SUPER^(); // FB_BA_View
Dst(); // FB_BA_BI_Raw
PlantLock(); // FB_BA_PlantLock
bPrioSfty := PlantLock.bPrioHigh OR PlantLock.bPrioLocalHigh;
bPrioCrit := PlantLock.bPrioMedium OR PlantLock.bPrioLocalMedium;
bDst := bPrioSfty OR bPrioCrit;
PrioSwiVal(
    bEn01 := stCmd.bEnSfty,
    nVal01 := stCmd.eValSfty,
    bEn02 := stCmd.bEnCrit,
    nVal02 := stCmd.eValCrit,
    bEn03 := stCmd.bEnPgm,
    nVal03 := stCmd.eValPgm); // FB_BA_PrioSwi_UDI04
MuxCmd(
    bEn := TRUE,
    nSel := PrioSwiVal.nVal,
    nEn01 := E_BA_Mdlt.eOff,
    bVal01 := FALSE,
    nEn02 := E_BA_Mdlt.eOn,
    bVal02 := TRUE,
    nEn03 := E_BA_Mdlt.eMin,
    bVal03 := TRUE,
    nEn04 := E_BA_Mdlt.eMax,
    bVal04 := TRUE); // FB_BA_MMUX_B04
Cmd(
    bEnSfty := stCmd.bEnSfty OR bPrioSfty,
    bValSfty := SEL(bPrioSfty, MuxCmd.bVal, FALSE),
    bEnCrit := stCmd.bEnCrit OR bPrioCrit,
    bValCrit := _w1,
    bEnPgm := stCmd.bEnPgm,
    bValPgm := MuxCmd.bVal); // FB_BA_BO_Raw
_w1 := SEL(bPrioCrit, MuxCmd.bVal, FALSE);
bCmd := Cmd.bPresentValue;
eActivePrio := Cmd.eActivePrio;
Ctrl(bEn := bCmd, fSetpoint := Sp.fPresentValue, fCtrlVal := fIn); // FB_BA_Loop
Sp(); // FB_BA_AV_Op
fMin := Ctrl.fMinOutputRm;
fMax := Ctrl.fMaxOutputRm;
MuxMdlt(
    bEn := bCmd,
    nSel := PrioSwiVal.nVal,
    nEn01 := E_BA_Mdlt.eOff,
    fVal01 := 0,
    nEn02 := E_BA_Mdlt.eOn,
    fVal02 := Ctrl.fPresentValue,
    nEn03 := E_BA_Mdlt.eMin,
    fVal03 := fMin,
    nEn04 := E_BA_Mdlt.eMax,
    fVal04 := fMax); // FB_BA_MMUX_R04
Mdlt(
    bEnSfty := Cmd.bEnSfty,
    fValSfty := SEL(bPrioSfty, MuxMdlt.fVal, 0),
    bEnCrit := Cmd.bEnCrit,
    fValCrit := _w2,
    bEnPgm := Cmd.bEnPgm,
    fValPgm := MuxMdlt.fVal); // FB_BA_AO_Raw
_w2 := SEL(bPrioCrit, MuxMdlt.fVal, 0);
fMdlt := Mdlt.fPresentValue;

METHOD FB_init : BOOL
VAR_INPUT
	bInitRetains : BOOL; // if TRUE, the retain variables are initialized (warm start / cold start)
	bInCopyCode : BOOL;  // if TRUE, the instance afterwards gets moved into the copy code (online change)
END_VAR
PlantLock.Parent					:= THIS^;		

Dst.iParent							:= THIS^;
Dst.iLabel							:= LblFun_Fault;  
Dst.ePolarity						:= E_BA_Polarity.eReverse;
Dst.sActiveText 					:= txtEvent_Triggered;
Dst.sInactiveText 					:= txtEvent_Normal;
Dst.nEventClassID					:= EC_ID.NC30;
Dst.stTimeDelay.nToNormal			:= BA2_Param.nDefTimeDelay_ToNormal;
Dst.stTimeDelay.nToAbnormal			:= BA2_Param.nDefTimeDelay_ToAbnormal;
Dst.bAlarmValue						:= TRUE;
Dst.aEventTransitionText[1]			:= txtEvent_Triggered;
Dst.aEventTransitionText[2]			:= txtEvent_Error;
Dst.aEventTransitionText[3]			:= txtEvent_Normal;
Dst.bEventDetectionEnable			:= TRUE;
Dst.eEnPlantLock					:= E_BA_LockPriority.eLocalMedium;

Cmd.iParent							:= THIS^;
Cmd.iLabel							:= LblFun_SwitchingCommand;  
Cmd.ePolarity						:= E_BA_Polarity.eNormal;
Cmd.sActiveText 					:= txtEvent_On;
Cmd.sInactiveText 					:= txtEvent_Off;
Cmd.bEnManualRm						:= FALSE;	//	Priority  8	
Cmd.bValManualRm					:= FALSE;	//	Priority  8
Cmd.nEventClassID					:= EC_ID.NC40;
Cmd.stTimeDelay.nToNormal			:= BA2_Param.nDefTimeDelay_ToNormal;
Cmd.stTimeDelay.nToAbnormal			:= BA2_Param.nDefTimeDelay_ToAbnormal;
Cmd.aEventTransitionText[1]			:= txtEvent_Disturb;
Cmd.aEventTransitionText[2]			:= txtEvent_None;
Cmd.aEventTransitionText[3]			:= txtEvent_Normal;
Cmd.bEventDetectionEnable			:= FALSE;
Cmd.eEnPlantLock					:= E_BA_LockPriority.eNoLock;

Mdlt.iParent						:= THIS^;
Mdlt.iLabel							:= LblFun_ControlSignal;  
Mdlt.eUnit							:= E_BA_Unit.eOther_Percent;
Mdlt.fResolution 					:= 0.003051851;
Mdlt.fScaleOffset 					:= 0;
Mdlt.fCOVIncrement					:= BA2_Param.fDefCOVIncrement;
Mdlt.bEnManualRm					:= FALSE;	//	Priority  8	
Mdlt.fValManualRm					:= 0.0;		//	Priority  8
Mdlt.nEventClassID					:= EC_ID.NC80;
Mdlt.stTimeDelay.nToNormal			:= BA2_Param.nDefTimeDelay_ToNormal;
Mdlt.stTimeDelay.nToAbnormal		:= BA2_Param.nDefTimeDelay_ToAbnormal;
Mdlt.stHighLimit.bEnable			:= FALSE;
Mdlt.stHighLimit.fValue				:= 0.0;		
Mdlt.stLowLimit.bEnable				:= FALSE;
Mdlt.stLowLimit.fValue				:= 0.0;
Mdlt.fLimitDeadband 				:= BA2_Param.fDefLimitDeadband;
Mdlt.aEventTransitionText[1]		:= txtEvent_Disturb;
Mdlt.aEventTransitionText[2]		:= txtEvent_None;
Mdlt.aEventTransitionText[3]		:= txtEvent_Normal;
Mdlt.bEventDetectionEnable			:= FALSE;
Mdlt.eEnPlantLock					:= E_BA_LockPriority.eNoLock;

Sp.iParent							:= THIS^;
Sp.iLabel							:= LblFun_Setpoint; 
Sp.eUnit 							:= E_BA_Unit.ePressure_Pascals;								 
Sp.fValueRm							:= 250;
Sp.fCOVIncrement					:= BA2_Param.fDefCOVIncrement;

Ctrl.iParent						:= THIS^;
Ctrl.iLabel							:= LblFun_LoopObject;  
Ctrl.eOpMode						:= E_BA_PIDMode.ePID;								 	 										 
Ctrl.eOutputUnit					:= E_BA_Unit.eOther_Percent;
Ctrl.eActionRm						:= E_BA_Action.eReverse;
Ctrl.fProportionalConstant			:= 0.01;
Ctrl.fIntegralConstant				:= 60;
Ctrl.fDerivativeConstant			:= 0;
Ctrl.fMaxOutputRm 					:= 100;
Ctrl.fMinOutputRm					:= 20;
Ctrl.fCOVIncrement					:= 0;
Ctrl.nDampConstant					:= 0;
Ctrl.fNeutralZone					:= 0;
END_METHOD

END_FUNCTION_BLOCK

// ---- Templates/POUs/Trade/AirConditioning/Aggregates/PreHeater/FB_BA_AC_PreHtr.TcPOU
{region '#Template'}
	{attribute 'Version' := '6.0.0.0'}
	{attribute 'Tags' := '"LCID": "1031", "Text": "AC, Aggregates, pre-heater"'}
	{attribute 'Tags' := '"LCID": "1033", "Text": "AC, Aggregates, pre-heater"'}
	{attribute 'Using' := '"Type": "Template", "URI": "Priority"'}		 
	{attribute 'Using' := '"Type": "Template", "URI": "BA2_Param"'}
	{attribute 'Using' := '"Type": "Template", "URI": "EC_ID"'}
	{attribute 'Description' := '"LCID": "1031", "Text": "Aggregat Vorerhitzer"'}
	{attribute 'Description' := '"LCID": "1033", "Text": "Aggregate pre-heater"'}
{endregion}
FUNCTION_BLOCK FB_BA_AC_PreHtr EXTENDS FB_BA_View
VAR_INPUT
	fSpTSuA					: REAL;
	fTSuA					: REAL;
	bSyncTSuACtrl			: BOOL;
	fSyncTSuACtrl			: REAL;	
	bDehumf					: BOOL;
	bSkipPreRinse			: BOOL; // Vorspülen überspringen // Skip pre-rinse
	fTWth					: REAL;
	bTWthLowLimit			: BOOL;
	bResetDehumf    		: BOOL;
END_VAR
VAR_OUTPUT
	bCmd					: BOOL;
	fPresentValue			: REAL;			
	bFrost					: BOOL;
	bPreRinseReady			: BOOL;  
	bActiveSeqCtrl			: BOOL;	
END_VAR
VAR_IN_OUT
	stTSeqLink				: ST_BA_SeqLink; // Sequenz Link Struktur // Sequence link structure	
	stAggregate				: ST_BA_Aggregate;	
END_VAR
VAR_INPUT CONSTANT PERSISTENT
	{attribute 'parameterCategory' := 'Behaviour'}
	fHysPuOn : REAL := 5.0;
	{attribute 'parameterCategory' := 'Behaviour'}
	fHysPuOff : REAL := 1.0;
END_VAR
VAR_INPUT CONSTANT
	TFl						: FB_BA_SensorAnalog;												
	TRt						: FB_BA_SensorAnalog;			
	TSuACtrl				: FB_BA_AC_PreHtrTSuACtrl;
	TRtCtrl					: FB_BA_AC_TRtCtrl;	
	TFrost					: FB_BA_SensorAnalog;																	
	TFrostPrtcCtrlAir		: FB_BA_PID_Sp;
	FrostThermostat			: FB_BA_SensorBinary;
	Vlv						: FB_BA_Vlv;
	Pu						: FB_BA_Pu1st;
	PlantLock				: FB_BA_PlantLock;			
	Aggregate				: FB_BA_Aggregate;																											 							
END_VAR
VAR
	bPrioSfty				: BOOL;
	bPrioCrit				: BOOL;		
	PrioSwiVal				: FB_BA_PrioSwi_B04;	
	
	HysPu					: FB_BA_Swi2P;
	SyncTSuACtrl			: FB_BA_RFTrig;
	SyncSeqCtrlIsActive		: FB_BA_RFTrig;
	PrioSwiSync				: FB_BA_PrioSwi_R04;	
END_VAR
VAR // added by the converter: edge detectors and wires of the graphical bodies
    _s1 : ST_BA_Analog;
    _s2 : ST_BA_Binary;
    _w1 : ANY;
    _w2 : BOOL;
END_VAR

SUPER^(); // FB_BA_View
Aggregate(bFdbUp := bPreRinseReady, stAggregate := stAggregate); // FB_BA_Aggregate
PlantLock(); // FB_BA_PlantLock
bPrioSfty := PlantLock.bPrioHigh OR PlantLock.bPrioLocalHigh;
bPrioCrit := PlantLock.bPrioMedium OR PlantLock.bPrioLocalMedium;
TFl(); // FB_BA_SensorAnalog
TRt(); // FB_BA_SensorAnalog
PrioSwiVal(
    bEn01 := Aggregate.arrPriorities[Priority.nLifeSafety],
    bVal01 := Aggregate.bValue,
    bEn02 := Aggregate.arrPriorities[Priority.nCritical],
    bVal02 := Aggregate.bValue,
    bEn03 := Aggregate.arrPriorities[Priority.nProgram],
    bVal03 := Aggregate.bValue); // FB_BA_PrioSwi_B04
SyncTSuACtrl(bValue := bSyncTSuACtrl); // FB_BA_RFTrig
SyncSeqCtrlIsActive(bValue := TSuACtrl.bSeqActv); // FB_BA_RFTrig
PrioSwiSync(
    bEn01 := SyncTSuACtrl.Qr,
    fVal01 := fSyncTSuACtrl,
    bEn04 := SyncSeqCtrlIsActive.Qr AND bActiveSeqCtrl AND bTWthLowLimit,
    fVal04 := Vlv.fMdlt); // FB_BA_PrioSwi_R04
TSuACtrl(
    bEn := PrioSwiVal.bVal,
    fSpTSuA := fSpTSuA,
    fTSuA := fTSuA,
    bSync := PrioSwiSync.bQ,
    fSync := PrioSwiSync.fVal,
    bDehumf := bDehumf,
    bResetDehumf := bResetDehumf,
    stSeqLink := stTSeqLink); // FB_BA_AC_PreHtrTSuACtrl
bActiveSeqCtrl := TSuACtrl.bIsActive;
TRtCtrl(
    bEnPreRinse := PrioSwiVal.bVal,
    fTRt := TRt.fPresentValue,
    bTWthLowLimit := bTWthLowLimit,
    fTWth := fTWth,
    bSkipPreRinse := bSkipPreRinse,
    bSeqActive := stTSeqLink.bEnSeqLink); // FB_BA_AC_TRtCtrl
bPreRinseReady := TRtCtrl.bPreRinseReady;
TFrost(); // FB_BA_SensorAnalog
TFrostPrtcCtrlAir(bEn := TRUE, fX := TFrost.fPresentValue); // FB_BA_PID_Sp
FrostThermostat(); // FB_BA_SensorBinary
bFrost := TFrost.eEventState = E_BA_EventState.eLowLimit OR FrostThermostat.bPresentValue;
_w1 := MAX(TSuACtrl.fY, TRtCtrl.fY, TFrostPrtcCtrlAir.fY);
// compose _s1 : ST_BA_Analog
_s1.bEnSfty := Aggregate.arrPriorities[Priority.nLifeSafety] OR bPrioSfty;
_s1.fValSfty := _w1;
_s1.bEnCrit := Aggregate.arrPriorities[Priority.nCritical] OR bPrioCrit OR bFrost;
_s1.fValCrit := SEL(bFrost, _w1, 100);
_s1.bEnPgm := TRUE;
_s1.fValPgm := _w1;
Vlv(stCmd := _s1); // FB_BA_Vlv
fPresentValue := Vlv.fMdlt;
HysPu(bEn := TRUE, fIn := fPresentValue, fOn := fHysPuOn, fOff := fHysPuOff); // FB_BA_Swi2P
_w2 := HysPu.bQ OR bTWthLowLimit OR bFrost;
// compose _s2 : ST_BA_Binary
_s2.bEnSfty := Vlv.stCmd.bEnSfty;
_s2.bValSfty := _w2;
_s2.bEnCrit := Vlv.stCmd.bEnCrit;
_s2.bValCrit := _w2;
_s2.bEnPgm := TRUE;
_s2.bValPgm := _w2;
Pu(stCmd := _s2); // FB_BA_Pu1st
bCmd := Pu.bCmd;

METHOD FB_init : BOOL
VAR_INPUT
	bInitRetains : BOOL; // if TRUE, the retain variables are initialized (warm start / cold start)
	bInCopyCode : BOOL;  // if TRUE, the instance afterwards gets moved into the copy code (online change)
END_VAR
PlantLock.Parent								:= THIS^;		

TFl.iParent										:= THIS^;		
TFl.iLabel										:= LblAgg_TemperatureFlow;   
TFl.sObjectName									:= '{Idx=11}';						 
TFl.eDPADMode									:= E_BA_DPADMode.eInclude;
TFl.MV.eUnit									:= E_BA_Unit.eTemperature_DegreesCelsius;
TFl.MV.fResolution 								:= 0.01;
TFl.MV.fScaleOffset 							:= 0; 
TFl.MV.bEventDetectionEnable					:= TRUE;
TFl.MV.eEnPlantLock								:= E_BA_LockPriority.eNoLock;
                            					                            					
TRt.iParent										:= THIS^;		
TRt.iLabel										:= LblAgg_TemperatureReturnFlow;   
TRt.sObjectName									:= '{Idx=11}';						 
TRt.eDPADMode									:= E_BA_DPADMode.eInclude;
TRt.MV.eUnit									:= E_BA_Unit.eTemperature_DegreesCelsius;
TRt.MV.fResolution 								:= 0.01;
TRt.MV.fScaleOffset 							:= 0;  
TRt.MV.bEventDetectionEnable					:= TRUE;
TRt.MV.eEnPlantLock								:= E_BA_LockPriority.eMedium;

TSuACtrl.iParent								:= THIS^;	
TSuACtrl.iLabel									:= LblCtl_SupplyAirTemperatureControl;   
TSuACtrl.sObjectName							:= '{Idx=11}';						 
TSuACtrl.eDPADMode								:= E_BA_DPADMode.eInclude;								

TRtCtrl.iParent									:= THIS^;
TRtCtrl.iLabel									:= LblCtl_ReturnWaterControl;   
TRtCtrl.sObjectName								:= '{Idx=12}';						 
TRtCtrl.eDPADMode								:= E_BA_DPADMode.eInclude;								
TRtCtrl.PreRinseDst.bEventDetectionEnable		:= TRUE;
TRtCtrl.PreRinseDst.eEnPlantLock				:= E_BA_LockPriority.eNoLock;
	                                				
TFrost.iParent									:= THIS^;		
TFrost.iLabel									:= LblCtl_TemperatureFrost;   
TFrost.sObjectName								:= '{Idx=11}';						 
TFrost.eDPADMode								:= E_BA_DPADMode.eInclude;
TFrost.MV.eUnit									:= E_BA_Unit.eTemperature_DegreesCelsius;
TFrost.MV.fResolution 							:= 0.0004577776;
TFrost.MV.fScaleOffset 							:= 0;  
TFrost.MV.bEventDetectionEnable					:= TRUE;
TFrost.MV.eEnPlantLock							:= E_BA_LockPriority.eMedium;

TFrostPrtcCtrlAir.iParent						:= THIS^;	
TFrostPrtcCtrlAir.iLabel						:= LblCtl_FrostProtectionControl;   
TFrostPrtcCtrlAir.sObjectName					:= '{Idx=13}';						 
TFrostPrtcCtrlAir.eDPADMode						:= E_BA_DPADMode.eInclude;
TFrostPrtcCtrlAir.Sp.fValueRm 					:= 5.0;
TFrostPrtcCtrlAir.Ctrl.fProportionalConstant	:= 5;
TFrostPrtcCtrlAir.Ctrl.fIntegralConstant		:= 60;	
TFrostPrtcCtrlAir.Ctrl.eActionRm				:= E_BA_Action.eReverse;

FrostThermostat.iParent							:= THIS^; 
FrostThermostat.iLabel							:= LblAgg_FrostProtectionMonitor;   
FrostThermostat.sObjectName						:= '{Idx=13}';						 
FrostThermostat.eDPADMode						:= E_BA_DPADMode.eInclude;
FrostThermostat.Input.iLabel					:= LblFun_OperationalMessage;   
FrostThermostat.Input.sObjectName				:= '{Idx=13}';						 
FrostThermostat.Input.ePolarity					:= E_BA_Polarity.eReverse;
FrostThermostat.Input.sActiveText 				:= txtEvent_Triggered;
FrostThermostat.Input.sInactiveText 			:= txtEvent_Normal;
FrostThermostat.Input.nEventClassID				:= EC_ID.NC30;
FrostThermostat.Input.aEventTransitionText[1]	:= txtEvent_Triggered;
FrostThermostat.Input.aEventTransitionText[2]	:= txtEvent_Error;
FrostThermostat.Input.aEventTransitionText[3]	:= txtEvent_Normal;
FrostThermostat.Input.bEventDetectionEnable		:= TRUE;
FrostThermostat.Input.eEnPlantLock				:= E_BA_LockPriority.eMedium;	

Vlv.iParent										:= THIS^;
Vlv.iLabel										:= LblAgg_Valve;    									 
Vlv.sObjectName									:= '{Idx=11}';						 
Vlv.eDPADMode									:= E_BA_DPADMode.eInclude;								
                            					
Pu.iParent										:= THIS^;
Pu.iLabel										:= LblAgg_Pump;   									 
Pu.sObjectName									:= '{Idx=11}';						 
Pu.eDPADMode									:= E_BA_DPADMode.eInclude;
Pu.Dst.bEventDetectionEnable					:= TRUE;
Pu.Dst.eEnPlantLock								:= E_BA_LockPriority.eMedium;
END_METHOD

END_FUNCTION_BLOCK

// ---- Templates/POUs/Universal/Pump/1st/FB_BA_Pu1st.TcPOU
{region '#Template'}
	{attribute 'Version' := '5.0.0.0'}
	{attribute 'Tags' := '"LCID": "1031", "Text": "Universal, Pump"'}
	{attribute 'Tags' := '"LCID": "1033", "Text": "Universal, Pump"'}
	{attribute 'Using' := '"Type": "Template", "URI": "EC_ID"'}
	{attribute 'Using' := '"Type": "Template", "URI": "BA2_Param"'}
	{attribute 'Description' := '"LCID": "1031", "Text": "Pumpe 1 stufig"'}
	{attribute 'Description' := '"LCID": "1033", "Text": "Pump 1 stage"'}
{endregion}	 
FUNCTION_BLOCK FB_BA_Pu1st EXTENDS FB_BA_Mot1st
VAR_INPUT
	bAblkLock				: BOOL;	
END_VAR
VAR_INPUT CONSTANT
	DlyOff					: FB_BA_DlyOff;								
	Ablk					: FB_BA_AntiBlocking;							
END_VAR
VAR
	PrioSwiPgm				: FB_BA_PrioSwi_B04;
	tonAblkLock				: TON;
END_VAR
VAR // added by the converter: edge detectors and wires of the graphical bodies
    _s1 : ST_BA_Binary;
END_VAR

DlyOff(bVal := stCmd.bEnPgm AND stCmd.bValPgm); // FB_BA_DlyOff
tonAblkLock(IN := bAblkLock, PT := T#2s); // TON
Ablk(bFdb := bCmd, bLock := tonAblkLock.Q); // FB_BA_AntiBlocking
PrioSwiPgm(bEn03 := DlyOff.bQ, bVal03 := TRUE, bEn04 := Ablk.bQ, bVal04 := TRUE); // FB_BA_PrioSwi_B04
// compose _s1 : ST_BA_Binary
_s1.bEnSfty := stCmd.bEnSfty;
_s1.bValSfty := stCmd.bValSfty;
_s1.bEnCrit := stCmd.bEnCrit;
_s1.bValCrit := stCmd.bValCrit;
_s1.bEnPgm := PrioSwiPgm.bQ;
_s1.bValPgm := PrioSwiPgm.bVal;
SUPER^(stCmd := _s1); // FB_BA_Mot1st

METHOD FB_init : BOOL
VAR_INPUT
	bInitRetains : BOOL; // if TRUE, the retain variables are initialized (warm start / cold start)
	bInCopyCode : BOOL;  // if TRUE, the instance afterwards gets moved into the copy code (online change)
END_VAR
DlyOff.iParent			:= THIS^;	
DlyOff.iLabel			:= LblCtl_DelayOff;
DlyOff.eDPADMode		:= E_BA_DPADMode.eIncludeDescription;

Ablk.iParent			:= THIS^;	 
Ablk.iLabel				:= LblCtl_AntiBlocking;
Ablk.eDPADMode			:= E_BA_DPADMode.eIncludeDescription;
END_METHOD

END_FUNCTION_BLOCK

// ---- Templates/POUs/Trade/AirConditioning/General/FB_BA_AC_OpMod1St.TcPOU
{region '#Template'}
	{attribute 'Version' := '6.0.0.0'}
	{attribute 'Tags' := '"LCID": "1031", "Text": "AC, Allgemein, AHU, Betriebsart"'}
	{attribute 'Tags' := '"LCID": "1033", "Text": "AC, General, AHU, Operating mode"'}
	{attribute 'Using' := '"Type": "Template", "URI": "E_BA_AC_OpMod01"'}
	{attribute 'Using' := '"Type": "Template", "URI": "E_BA_OnOffA"'}
	{attribute 'Using' := '"Type": "Template", "URI": "E_BA_OnOff"'}
	{attribute 'Description' := '"LCID": "1031", "Text": "Betriebsart"'}
	{attribute 'Description' := '"LCID": "1033", "Text": "Operating mode"'}
{endregion}
FUNCTION_BLOCK FB_BA_AC_OpMod1St EXTENDS FB_BA_View
VAR_INPUT
	bSmExtt					: BOOL;	// smoke extraction 
	bFireDetc				: BOOL;	// fire detection alarm
	bForcVent				: BOOL;	// Forced ventilation
	bEmgOff					: BOOL;	// emergency stop
	bFrst					: BOOL;	// Frost protection is active
	bCentSwiOff				: BOOL;	// Central switch-off	
	bAlmShutOff				: BOOL;	// Shut Off plant collective alarm
	bNgtCol					: BOOL;	// Summer night cooling
	bColDwnPrtc				: BOOL;	// Cooling down protection
	bOvrHtgPrtc				: BOOL;	// Overheating protection
END_VAR
VAR_OUTPUT
	eOpMode					: E_BA_AC_OpMod01;
END_VAR
VAR_INPUT CONSTANT
	OpModMan				: FB_BA_MV_Op;	
	Sched					: FB_BA_SchedM;
	OpModPr					: FB_BA_MV_Op;
END_VAR
VAR
	PrioSwiOpMod			: FB_BA_PrioSwi_UDI24;
END_VAR

SUPER^(); // FB_BA_View
OpModMan(); // FB_BA_MV_Op
Sched(); // FB_BA_SchedM
PrioSwiOpMod(
    bEn02 := bSmExtt,
    nVal02 := E_BA_AC_OpMod01.eSmokeExtractionProgram,
    bEn04 := bFireDetc,
    nVal04 := E_BA_AC_OpMod01.eFire,
    bEn05 := bCentSwiOff,
    nVal05 := E_BA_AC_OpMod01.eCentralSwitchOff,
    bEn07 := bForcVent,
    nVal07 := E_BA_AC_OpMod01.eForcedVentilation,
    bEn08 := bEmgOff,
    nVal08 := E_BA_AC_OpMod01.eEmergency,
    bEn09 := bFrst,
    nVal09 := E_BA_AC_OpMod01.eFrost,
    bEn10 := bAlmShutOff,
    nVal10 := E_BA_AC_OpMod01.eAlarm,
    bEn14 := E_BA_OnOffA.eOff = OpModMan.nPresentValue,
    nVal14 := E_BA_AC_OpMod01.eOff,
    bEn15 := OpModMan.nPresentValue = E_BA_OnOffA.eOn,
    nVal15 := E_BA_AC_OpMod01.eOn,
    bEn18 := Sched.nPresentValue = E_BA_OnOff.eOn,
    nVal18 := E_BA_AC_OpMod01.eOn,
    bEn20 := bNgtCol,
    nVal20 := E_BA_AC_OpMod01.eNightCooling,
    bEn21 := bColDwnPrtc,
    nVal21 := E_BA_AC_OpMod01.eCoolDownProtection,
    bEn22 := bOvrHtgPrtc,
    nVal22 := E_BA_AC_OpMod01.eOverHeatingProtection,
    bEn24 := TRUE,
    nVal24 := E_BA_AC_OpMod01.eOFF); // FB_BA_PrioSwi_UDI24
OpModPr(nValuePgm := PrioSwiOpMod.nVal); // FB_BA_MV_Op
eOpMode := OpModPr.nPresentValue;

METHOD FB_init : BOOL
VAR_INPUT
	bInitRetains : BOOL; // if TRUE, the retain variables are initialized (warm start / cold start)
	bInCopyCode : BOOL;  // if TRUE, the instance afterwards gets moved into the copy code (online change)
END_VAR
OpModMan.iParent			:= THIS^;
OpModMan.iLabel				:= LblCtl_OperationModeSelection; 	
OpModMan.aStateText[1]		:= txtEvent_Auto;
OpModMan.aStateText[2]		:= txtEvent_Off;
OpModMan.aStateText[3]		:= txtEvent_On;
OpModMan.nValueRm			:= E_BA_OnOffA.eAutomatic;

OpModPr.iParent				:= THIS^;
OpModPr.iLabel				:= LblCtl_PresentOperationMode; 								 	 
OpModPr.aStateText[1]		:= txtEvent_Off;
OpModPr.aStateText[2]		:= txtEvent_On;
OpModPr.aStateText[3]		:= txtEvent_EmergencyStop;
OpModPr.aStateText[4]		:= txtEvent_Frost;
OpModPr.aStateText[5]		:= txtEvent_SmokeExtraction_P;
OpModPr.aStateText[6]		:= txtEvent_SmokeExtractionSupplyAir;
OpModPr.aStateText[7]		:= txtEvent_SmokeExtractionExtractAir;
OpModPr.aStateText[8]		:= txtEvent_Fire;
OpModPr.aStateText[9]		:= txtEvent_NightCooling;
OpModPr.aStateText[10]		:= txtEvent_CoolDownProtection;
OpModPr.aStateText[11]		:= txtEvent_OverHeatingProtection;
OpModPr.aStateText[12]		:= txtEvent_Disturb;
OpModPr.aStateText[13]		:= txtEvent_ForcedVentilation;
OpModPr.aStateText[14]		:= txtEvent_CentralSwitchOff; 		

Sched.iParent											:= THIS^;
Sched.iLabel											:= LblFun_Scheduler; 			
Sched.aStateText[1]										:= txtEvent_Off;
Sched.aStateText[2]										:= txtEvent_On;
Sched.nPredictTime										:= 0;
Sched.nDefaultValue										:= E_BA_OnOff.eOff;
Sched.bWriteWeekly										:= FALSE;
//	Monday
Sched.aWeek[E_BA_Weekday.eMonday,1].eState				:= E_BA_SchedEntryState.eValue;
Sched.aWeek[E_BA_Weekday.eMonday,1].uValue.udiVal		:= E_BA_OnOff.eOn;
Sched.aWeek[E_BA_Weekday.eMonday,1].stTime.nHour		:= 6;
Sched.aWeek[E_BA_Weekday.eMonday,1].stTime.nMinute		:= 0;
Sched.aWeek[E_BA_Weekday.eMonday,1].stTime.nSecond		:= 0;
Sched.aWeek[E_BA_Weekday.eMonday,2].eState				:= E_BA_SchedEntryState.eValue;
Sched.aWeek[E_BA_Weekday.eMonday,2].uValue.udiVal		:= E_BA_OnOff.eOff;
Sched.aWeek[E_BA_Weekday.eMonday,2].stTime.nHour		:= 20;
Sched.aWeek[E_BA_Weekday.eMonday,2].stTime.nMinute		:= 0;
Sched.aWeek[E_BA_Weekday.eMonday,2].stTime.nSecond		:= 0;
Sched.aWeek[E_BA_Weekday.eMonday,3].eState				:= E_BA_SchedEntryState.eValue;
Sched.aWeek[E_BA_Weekday.eMonday,3].uValue.udiVal		:= E_BA_OnOff.eOff;
Sched.aWeek[E_BA_Weekday.eMonday,3].stTime.nHour		:= 0;
Sched.aWeek[E_BA_Weekday.eMonday,3].stTime.nMinute		:= 0;
Sched.aWeek[E_BA_Weekday.eMonday,3].stTime.nSecond		:= 0;
//	Tuesday
Sched.aWeek[E_BA_Weekday.eTuesday,1].eState				:= E_BA_SchedEntryState.eValue;
Sched.aWeek[E_BA_Weekday.eTuesday,1].uValue.udiVal		:= E_BA_OnOff.eOn;
Sched.aWeek[E_BA_Weekday.eTuesday,1].stTime.nHour		:= 6;
Sched.aWeek[E_BA_Weekday.eTuesday,1].stTime.nMinute		:= 0;
Sched.aWeek[E_BA_Weekday.eTuesday,1].stTime.nSecond		:= 0;
Sched.aWeek[E_BA_Weekday.eTuesday,2].eState				:= E_BA_SchedEntryState.eValue;
Sched.aWeek[E_BA_Weekday.eTuesday,2].uValue.udiVal		:= E_BA_OnOff.eOff;
Sched.aWeek[E_BA_Weekday.eTuesday,2].stTime.nHour		:= 20;
Sched.aWeek[E_BA_Weekday.eTuesday,2].stTime.nMinute		:= 0;
Sched.aWeek[E_BA_Weekday.eTuesday,2].stTime.nSecond		:= 0;
Sched.aWeek[E_BA_Weekday.eTuesday,3].eState				:= E_BA_SchedEntryState.eValue;
Sched.aWeek[E_BA_Weekday.eTuesday,3].uValue.udiVal		:= E_BA_OnOff.eOff;
Sched.aWeek[E_BA_Weekday.eTuesday,3].stTime.nHour		:= 0;
Sched.aWeek[E_BA_Weekday.eTuesday,3].stTime.nMinute		:= 0;
Sched.aWeek[E_BA_Weekday.eTuesday,3].stTime.nSecond		:= 0;
//	Wednesday
Sched.aWeek[E_BA_Weekday.eWednesday,1].eState			:= E_BA_SchedEntryState.eValue;
Sched.aWeek[E_BA_Weekday.eWednesday,1].uValue.udiVal	:= E_BA_OnOff.eOn;
Sched.aWeek[E_BA_Weekday.eWednesday,1].stTime.nHour		:= 6;
Sched.aWeek[E_BA_Weekday.eWednesday,1].stTime.nMinute	:= 0;
Sched.aWeek[E_BA_Weekday.eWednesday,1].stTime.nSecond	:= 0;
Sched.aWeek[E_BA_Weekday.eWednesday,2].eState			:= E_BA_SchedEntryState.eValue;
Sched.aWeek[E_BA_Weekday.eWednesday,2].uValue.udiVal	:= E_BA_OnOff.eOff;
Sched.aWeek[E_BA_Weekday.eWednesday,2].stTime.nHour		:= 20;
Sched.aWeek[E_BA_Weekday.eWednesday,2].stTime.nMinute	:= 0;
Sched.aWeek[E_BA_Weekday.eWednesday,2].stTime.nSecond	:= 0;
Sched.aWeek[E_BA_Weekday.eWednesday,3].eState			:= E_BA_SchedEntryState.eValue;
Sched.aWeek[E_BA_Weekday.eWednesday,3].uValue.udiVal	:= E_BA_OnOff.eOff;
Sched.aWeek[E_BA_Weekday.eWednesday,3].stTime.nHour		:= 0;
Sched.aWeek[E_BA_Weekday.eWednesday,3].stTime.nMinute	:= 0;
Sched.aWeek[E_BA_Weekday.eWednesday,3].stTime.nSecond	:= 0;
//	Thursday
Sched.aWeek[E_BA_Weekday.eThursday,1].eState			:= E_BA_SchedEntryState.eValue;
Sched.aWeek[E_BA_Weekday.eThursday,1].uValue.udiVal		:= E_BA_OnOff.eOn;
Sched.aWeek[E_BA_Weekday.eThursday,1].stTime.nHour		:= 6;
Sched.aWeek[E_BA_Weekday.eThursday,1].stTime.nMinute	:= 0;
Sched.aWeek[E_BA_Weekday.eThursday,1].stTime.nSecond	:= 0;
Sched.aWeek[E_BA_Weekday.eThursday,2].eState			:= E_BA_SchedEntryState.eValue;
Sched.aWeek[E_BA_Weekday.eThursday,2].uValue.udiVal		:= E_BA_OnOff.eOff;
Sched.aWeek[E_BA_Weekday.eThursday,2].stTime.nHour		:= 20;
Sched.aWeek[E_BA_Weekday.eThursday,2].stTime.nMinute	:= 0;
Sched.aWeek[E_BA_Weekday.eThursday,2].stTime.nSecond	:= 0;
Sched.aWeek[E_BA_Weekday.eThursday,3].eState			:= E_BA_SchedEntryState.eValue;
Sched.aWeek[E_BA_Weekday.eThursday,3].uValue.udiVal		:= E_BA_OnOff.eOff;
Sched.aWeek[E_BA_Weekday.eThursday,3].stTime.nHour		:= 0;
Sched.aWeek[E_BA_Weekday.eThursday,3].stTime.nMinute	:= 0;
Sched.aWeek[E_BA_Weekday.eThursday,3].stTime.nSecond	:= 0;
//	Friday
Sched.aWeek[E_BA_Weekday.eFriday,1].eState				:= E_BA_SchedEntryState.eValue;
Sched.aWeek[E_BA_Weekday.eFriday,1].uValue.udiVal		:= E_BA_OnOff.eOn;
Sched.aWeek[E_BA_Weekday.eFriday,1].stTime.nHour		:= 6;
Sched.aWeek[E_BA_Weekday.eFriday,1].stTime.nMinute		:= 0;
Sched.aWeek[E_BA_Weekday.eFriday,1].stTime.nSecond		:= 0;
Sched.aWeek[E_BA_Weekday.eFriday,2].eState				:= E_BA_SchedEntryState.eValue;
Sched.aWeek[E_BA_Weekday.eFriday,2].uValue.udiVal		:= E_BA_OnOff.eOff;
Sched.aWeek[E_BA_Weekday.eFriday,2].stTime.nHour		:= 20;
Sched.aWeek[E_BA_Weekday.eFriday,2].stTime.nMinute		:= 0;
Sched.aWeek[E_BA_Weekday.eFriday,2].stTime.nSecond		:= 0;
Sched.aWeek[E_BA_Weekday.eFriday,3].eState				:= E_BA_SchedEntryState.eValue;
Sched.aWeek[E_BA_Weekday.eFriday,3].uValue.udiVal		:= E_BA_OnOff.eOff;
Sched.aWeek[E_BA_Weekday.eFriday,3].stTime.nHour		:= 0;
Sched.aWeek[E_BA_Weekday.eFriday,3].stTime.nMinute		:= 0;
Sched.aWeek[E_BA_Weekday.eFriday,3].stTime.nSecond		:= 0;
Sched.bWriteException									:= FALSE;
END_METHOD

END_FUNCTION_BLOCK

// ---- Templates/POUs/Trade/AutomationControl/ControlCabinet/FB_BA_ControlCabinet.TcPOU
{region '#Template'}
	{attribute 'Version' := '5.0.1.0'}
	{attribute 'Tags' := '"LCID": "1031", "Text": "General, Cabinet, Control cabinet"'}
	{attribute 'Tags' := '"LCID": "1033", "Text": "General, Cabinet, Control cabinet"'}
	{attribute 'Using' := '"Type": "Template", "URI": "EC_ID"'}
	{attribute 'Description' := '"LCID": "1031", "Text": "Schaltschrank Ereignisse"'}
	{attribute 'Description' := '"LCID": "1033", "Text": "Control cabinet events"'}
{endregion}
FUNCTION_BLOCK FB_BA_ControlCabinet EXTENDS FB_BA_ControlCabinetBasic
VAR_INPUT CONSTANT
	Fuse01					: FB_BA_SensorBinary;		
	Fuse02					: FB_BA_SensorBinary;	
	Fuse03					: FB_BA_SensorBinary;	
END_VAR

SUPER^(); // FB_BA_ControlCabinetBasic
Fuse01(); // FB_BA_SensorBinary
Fuse02(); // FB_BA_SensorBinary
Fuse03(); // FB_BA_SensorBinary

METHOD FB_init : BOOL
VAR_INPUT
	bInitRetains : BOOL; // if TRUE, the retain variables are initialized (warm start / cold start)
	bInCopyCode : BOOL;  // if TRUE, the instance afterwards gets moved into the copy code (online change)
END_VAR
Fuse01.iParent								:= THIS^;
Fuse01.iLabel								:= LblCtl_Fuse;
Fuse01.sObjectName							:='{Idx=10}';	
Fuse01.eDPADMode							:= E_BA_DPADMode.eInclude;	
Fuse01.Input.iLabel							:= LblFun_Fault;																																									
Fuse01.Input.ePolarity						:= E_BA_Polarity.eReverse;
Fuse01.Input.sActiveText 					:= txtEvent_Triggered;
Fuse01.Input.sInactiveText 					:= txtEvent_Normal;
Fuse01.Input.nEventClassID					:= EC_ID.NC30;
Fuse01.Input.aEventTransitionText[1]		:= txtEvent_Triggered;
Fuse01.Input.aEventTransitionText[2]		:= txtEvent_Error;
Fuse01.Input.aEventTransitionText[3]		:= txtEvent_Normal;
Fuse01.Input.bEventDetectionEnable			:= TRUE;

Fuse01.Input.eEnPlantLock					:= E_BA_LockPriority.eNoLock;	
								 
Fuse02.iParent								:= THIS^;		
Fuse02.iLabel								:= LblCtl_Fuse;	
Fuse02.sObjectName							:='{Idx=20}';	
Fuse02.eDPADMode							:= E_BA_DPADMode.eInclude;	
Fuse02.Input.iLabel							:= LblFun_Fault;																				
Fuse02.Input.ePolarity						:= E_BA_Polarity.eReverse;
Fuse02.Input.sActiveText 					:= txtEvent_Triggered;
Fuse02.Input.sInactiveText 					:= txtEvent_Normal;
Fuse02.Input.nEventClassID					:= EC_ID.NC30;
Fuse02.Input.aEventTransitionText[1]		:= txtEvent_Triggered;
Fuse02.Input.aEventTransitionText[2]		:= txtEvent_Error;
Fuse02.Input.aEventTransitionText[3]		:= txtEvent_Normal;
Fuse02.Input.bEventDetectionEnable			:= TRUE;

Fuse02.Input.eEnPlantLock					:= E_BA_LockPriority.eNoLock;	
										 
Fuse03.iParent								:= THIS^;		
Fuse03.iLabel								:= LblCtl_Fuse;	
Fuse03.sObjectName							:='{Idx=30}';	
Fuse03.eDPADMode							:= E_BA_DPADMode.eInclude;				
Fuse03.Input.iLabel							:= LblFun_Fault;																				
Fuse03.Input.ePolarity						:= E_BA_Polarity.eReverse;
Fuse03.Input.sActiveText 					:= txtEvent_Triggered;
Fuse03.Input.sInactiveText 					:= txtEvent_Normal;
Fuse03.Input.nEventClassID					:= EC_ID.NC30;
Fuse03.Input.aEventTransitionText[1]		:= txtEvent_Triggered;
Fuse03.Input.aEventTransitionText[2]		:= txtEvent_Error;
Fuse03.Input.aEventTransitionText[3]		:= txtEvent_Normal;
Fuse03.Input.bEventDetectionEnable			:= TRUE;

Fuse03.Input.eEnPlantLock					:= E_BA_LockPriority.eNoLock;
END_METHOD

END_FUNCTION_BLOCK

// ---- Templates/POUs/Trade/AutomationControl/Device/FB_BA_Device.TcPOU
{region '#Template'}
	{attribute 'Version' := '5.0.1.0'}
	{attribute 'Tags' := '"LCID": "1031", "Text": "Automatisierungssteuerung, Gerät, Einstellungen, Projekt, Parameter, Trend, Empfängerliste"'}
	{attribute 'Tags' := '"LCID": "1033", "Text": "Automation control, Device, Settings, Project, Parameter, Trend, Recipient list"'}
	{attribute 'Description' := '"LCID": "1031", "Text": "Basis Einstellungen der Steuerung"'}
	{attribute 'Description' := '"LCID": "1033", "Text": "Basic settings of the control"'}
{endregion}
	 
FUNCTION_BLOCK FB_BA_Device EXTENDS FB_BA_View
VAR_INPUT
END_VAR
VAR_INPUT CONSTANT
	Trend				: FB_BA_TrendLogging;	
	Project				: FB_BA_ProjectEx;
	Parameter			: FB_BA_Parameter;	
END_VAR
VAR_OUTPUT
END_VAR
VAR
	tonDlyStartPLC		: TON;	
END_VAR

SUPER^(); // FB_BA_View
tonDlyStartPLC(IN := TRUE, PT := T#2000ms); // TON
BA2_Param.bDlyStartPLC := tonDlyStartPLC.Q;
Parameter(); // FB_BA_Parameter
Trend(); // FB_BA_TrendLogging
// connect a UPS-monitoring FB at this input
Project(); // FB_BA_ProjectEx

METHOD FB_init : BOOL
VAR_INPUT
	bInitRetains : BOOL; // if TRUE, the retain variables are initialized (warm start / cold start)
	bInCopyCode : BOOL;  // if TRUE, the instance afterwards gets moved into the copy code (online change)
END_VAR
Project.iParent						:= THIS^;
Project.iLabel						:= LblComp_Project;
Project.sObjectName					:= '{Idx=11,Idx=99}';
Project.tPrsData_DefaultPeriod 		:= T#30M;
Project.tPrsData_ComissioningPeriod := T#10M;

Trend.iParent						:= THIS^;
Trend.iLabel						:= LblCtl_TrendLogging;
Trend.eDPADMode						:= E_BA_DPADMode.eInclude;
END_METHOD

END_FUNCTION_BLOCK

// ---- Templates/POUs/Universal/Control/Trend/FB_BA_TrendLogging.TcPOU
{region '#Template'}
	{attribute 'Version' := '5.0.1.0'}
	{attribute 'Tags' := '"LCID": "1031", "Text": "Universal, Control, Trend"'}
	{attribute 'Tags' := '"LCID": "1033", "Text": "Universal, Control, Trend"'}
	{attribute 'Using' := '"Type": "Template", "URI": "EC_ID"'}
	{attribute 'Using' := '"Type": "Template", "URI": "BA2_Param"'}
	{attribute 'Description' := '"LCID": "1031", "Text": "Trend"'}
	{attribute 'Description' := '"LCID": "1033", "Text": "Trend"'}
{endregion}			 
FUNCTION_BLOCK FB_BA_TrendLogging EXTENDS FB_BA_View
VAR_INPUT
END_VAR
VAR_OUTPUT
END_VAR
VAR_INPUT CONSTANT
	Trends						: ARRAY[1..TREND_COUNT] OF FB_BA_Trend;								
END_VAR
VAR
	i							: UDINT;
END_VAR
VAR CONSTANT
	TREND_COUNT						: UDINT := 30;
END_VAR

SUPER^();

FOR i := 1 TO TREND_COUNT DO
	Trends[i]();
END_FOR

METHOD FB_init : BOOL
VAR_INPUT
	bInitRetains : BOOL; // if TRUE, the retain variables are initialized (warm start / cold start)
	bInCopyCode : BOOL;  // if TRUE, the instance afterwards gets moved into the copy code (online change)
END_VAR 
VAR
END_VAR
FOR i := 1 TO TREND_COUNT DO
	Trends[i].iParent					:= THIS^;
	Trends[i].iLabel					:= LblFun_ObjectTrendLog;
	Trends[i].bEnable					:= BA2_Param.bTrend_DefLogEnable;
	Trends[i].stStartTime				:= BA2_Param.stTrend_DefStartTime;
	Trends[i].stStopTime				:= BA2_Param.stTrend_DefStopTime;	
	Trends[i].nLogInterval 				:= BA2_Param.nTrend_DefLogInterval;
	Trends[i].bStopOnFull				:= BA2_Param.bTrend_DefStopOnFull;
	Trends[i].nBufferSize 				:= BA2_Param.nTrend_BufferSize;
	Trends[i].eLoggingType				:= BA2_Param.eTrend_DefLoggingType;	
	Trends[i].nEventClassID				:= EC_ID.NC80;
	Trends[i].nNotificationThreshold	:= BA2_Param.nTrend_DefNotificationThreshold;
	Trends[i].aEventTransitionText[1]	:= txtEvent_Offnormal;
	Trends[i].aEventTransitionText[2]	:= txtEvent_None;
	Trends[i].aEventTransitionText[3]	:= txtEvent_Normal;
	Trends[i].bEventDetectionEnable		:= FALSE;
END_FOR
END_METHOD

END_FUNCTION_BLOCK

// ---- Templates/POUs/Trade/AutomationControl/Device/Project/FB_BA_ProjectEx.TcPOU
{region '#Template'}
	{attribute 'Version' := '5.0.0.0'}
	{attribute 'Tags' := '"LCID": "1031", "Text": "Automatisierungssteuerung, Gerät, Einstellungen, Projekt"'}
	{attribute 'Tags' := '"LCID": "1033", "Text": "Automation control, Device, Settings, Project"'}
	{attribute 'Description' := '"LCID": "1031", "Text": "Projektspezifische Informationen"'}
	{attribute 'Description' := '"LCID": "1033", "Text": "Project specific informations"'}
{endregion}
	 
FUNCTION_BLOCK FB_BA_ProjectEx EXTENDS FB_BA_Project
VAR_INPUT CONSTANT PERSISTENT
	{attribute 'parameterCategory' := 'Persistent Data'}
	tPrsData_DefaultPeriod : TIME := T#30M;
	{attribute 'parameterCategory' := 'Persistent Data'}
	tPrsData_ComissioningPeriod : TIME := T#10M;
END_VAR
VAR_INPUT CONSTANT
	{attribute 'parameterCategory' := 'Persistent Data'}
	bPrsData_ManualWriteData : BOOL;
END_VAR
VAR_INPUT
	bWrtPrsOnPowerFail		: BOOL;
END_VAR
VAR_OUTPUT
	nPrsDataWritten			: UINT;
END_VAR

SUPER^();

OnInitCycle();
PersistentData();

{attribute 'hide'}
METHOD PROTECTED OnInitCycle
VAR
	_stVersion		: ST_LibVersion;
END_VAR
VAR CONSTANT
	FORMAT			: STRING		:= '%d.%d.%d.%d';
END_VAR
CASE (State) OF
	E_BA_ObjectState.eInstanceInit1:
		// Refresh runtime information:
		{IF defined (pou: F_GetVersion)}
			_stVersion := F_GetVersion();
			
			XBA_Globals.FormatStr2(
				pFormatString := ADR(FORMAT),
				arg1:=F_UINT(_stVersion.iMajor),
				arg2:=F_UINT(_stVersion.iMinor),
				arg3:=F_UINT(_stVersion.iBuild),
				arg4:=F_UINT(_stVersion.iRevision),
			
				pDstString := ADR(fbDiag.stVersion.Project),
				nDstSize := SIZEOF(fbDiag.stVersion.Project)
			);
		{END_IF}
		
END_CASE
END_METHOD

{attribute 'hide'}
METHOD PROTECTED PersistentData
VAR_INST
	nOnlineChangeCnt		:	UDINT;
	iStep					:	INT;
	fbTon					:	TON;
	fbResetOnlineChange		:	TON;
	rtigManual				:	R_TRIG;
	trigUPS					:	R_TRIG;
	rFinishTrig				:	R_TRIG;
	WrtPersistDat			:	FB_BA_WrtPersistDat;
END_VAR
VAR CONSTANT
	DETECT_COMISSIONING_DURATION : TIME := T#60M;
END_VAR
IF	TwinCAT_SystemInfoVarList._AppInfo.OnlineChangeCnt <> nOnlineChangeCnt THEN
	nOnlineChangeCnt := TwinCAT_SystemInfoVarList._AppInfo.OnlineChangeCnt;
	fbResetOnlineChange(IN := FALSE);
	fbTon(IN := FALSE);
	iStep := 10;
END_IF

IF	tPrsData_DefaultPeriod < T#600S THEN
	tPrsData_DefaultPeriod	:= T#1800S;
END_IF

IF	tPrsData_ComissioningPeriod < T#30S THEN
	tPrsData_ComissioningPeriod	:= T#300S;
END_IF

CASE	iStep	OF
	0:
		fbTon(IN := NOT fbTon.Q,PT := tPrsData_DefaultPeriod);
	10:
		fbTon(IN := NOT fbTon.Q,PT := tPrsData_ComissioningPeriod);
		fbResetOnlineChange(IN := TRUE, PT := DETECT_COMISSIONING_DURATION);
		
		IF	fbResetOnlineChange.Q THEN
			iStep := 0;
			fbResetOnlineChange(IN := FALSE);
		END_IF
END_CASE
 
rtigManual(CLK := bPrsData_ManualWriteData);
bPrsData_ManualWriteData := FALSE;

trigUPS(CLK := bWrtPrsOnPowerFail);

// Write persistent data:
WrtPersistDat(bStt:=(fbTon.Q OR rtigManual.Q OR trigUPS.Q));
rFinishTrig(CLK:=(WrtPersistDat.bBusy AND NOT WrtPersistDat.bErr));

IF (rFinishTrig.Q) THEN
	nPrsDataWritten := (nPrsDataWritten+1);
END_IF
END_METHOD

END_FUNCTION_BLOCK

// ---- Templates/POUs/Trade/AutomationControl/EventClasses/FB_BA_EvtGroups.TcPOU
{region '#Template'}
	{attribute 'Version' := '5.0.0.0'}
	{attribute 'Tags' := '"LCID": "1031", "Text": "General, Cabinet, Control cabinet, Event groups, Categories, Notification classes, Event classes"'}
	{attribute 'Tags' := '"LCID": "1033", "Text": "General, Cabinet, Control cabinet, Event groups, Categories, Notification classes, Event classes"'}
	{attribute 'Using' := '"Type": "Template", "URI": "EC_ID"'}
	{attribute 'Description' := '"LCID": "1031", "Text": "Ereignisgruppen, Kategorien"'}
	{attribute 'Description' := '"LCID": "1033", "Text": "Event groups, categories"'}
{endregion}
FUNCTION_BLOCK FB_BA_EvtGroups EXTENDS FB_BA_View
VAR_INPUT CONSTANT
	LifeSafety						: FB_BA_EvtCategory;
	SafetyMsg						: FB_BA_EvtCategory;
	AlarmMsg						: FB_BA_EvtCategory;
	FaultMsg						: FB_BA_EvtCategory;
	MaintenanceMsg01				: FB_BA_EvtCategory;
	MaintenanceMsg02				: FB_BA_EvtCategory;
	SystemMsg						: FB_BA_EvtCategory;
	ManualOp						: FB_BA_EvtCategory;
	OtherMsg						: FB_BA_EvtCategory;
END_VAR

SUPER^(); // FB_BA_View
LifeSafety(); // FB_BA_EvtCategory
SafetyMsg(); // FB_BA_EvtCategory
AlarmMsg(); // FB_BA_EvtCategory
FaultMsg(); // FB_BA_EvtCategory
MaintenanceMsg01(); // FB_BA_EvtCategory
MaintenanceMsg02(); // FB_BA_EvtCategory
SystemMsg(); // FB_BA_EvtCategory
ManualOp(); // FB_BA_EvtCategory
OtherMsg(); // FB_BA_EvtCategory

METHOD FB_init : BOOL
VAR_INPUT
	bInitRetains : BOOL; // if TRUE, the retain variables are initialized (warm start / cold start)
	bInCopyCode : BOOL;  // if TRUE, the instance afterwards gets moved into the copy code (online change)
END_VAR
//===================================================================
// Ereigniskategorie - Gefahr für Leben // Event category - Danger to life
// Brandalarm, Überfall // Fire alarm, robbery
LifeSafety.iParent							:= THIS^;
LifeSafety.iLabel							:= LblCtl_EvtCategoryLifeSafty;
LifeSafety.eDPADMode						:= E_BA_DPADMode.eInclude;																						
LifeSafety.EC.nInstanceID					:= EC_ID.NC10;
LifeSafety.EC.iLabel						:= LblFun_ObjectNotificationClass;
LifeSafety.EC.sObjectName					:='{Idx=10}';
LifeSafety.EC.eAlarmMode					:= E_BA_AlarmMode.UserDefined;
LifeSafety.EC.eEventType					:= E_BA_EventType.eAlarm;
LifeSafety.EC.aPriority[1]					:= 10;
LifeSafety.EC.aPriority[2]					:= 11;
LifeSafety.EC.aPriority[3]					:= 12;
LifeSafety.EC.aAcknowledgeRequired[1]		:= TRUE;
LifeSafety.EC.aAcknowledgeRequired[2]		:= FALSE;
LifeSafety.EC.aAcknowledgeRequired[3]		:= TRUE;
//===================================================================		
// Ereigniskategorie - Gefahrenmeldung, Sicherheitsmeldung // Event category - hazard alert, safety message
// Einbruch, unberechtigter Zutritt // Burglary, unauthorised entry
SafetyMsg.iParent							:= THIS^;
SafetyMsg.iLabel							:= LblCtl_EvtCategorySaftyMessage;
SafetyMsg.eDPADMode							:= E_BA_DPADMode.eInclude;																						
SafetyMsg.EC.nInstanceID					:= EC_ID.NC20;
SafetyMsg.EC.iLabel							:= LblFun_ObjectNotificationClass;
SafetyMsg.EC.sObjectName					:='{Idx=20}';
SafetyMsg.EC.eAlarmMode						:= E_BA_AlarmMode.UserDefined;
SafetyMsg.EC.eEventType						:= E_BA_EventType.eAlarm;
SafetyMsg.EC.aPriority[1]					:= 40;
SafetyMsg.EC.aPriority[2]					:= 41;
SafetyMsg.EC.aPriority[3]					:= 42;
SafetyMsg.EC.aAcknowledgeRequired[1]		:= TRUE;
SafetyMsg.EC.aAcknowledgeRequired[2]		:= FALSE;
SafetyMsg.EC.aAcknowledgeRequired[3]		:= TRUE;
//===================================================================//
// Ereigniskategorie - Alarmeldung - Meldung signalisiert Anlagenausfall oder erfordert sofortigen Eingriff 
// Event category - Alarm message - Message signals system failure or requires immediate intervention 
// Sicherheitstemperaturbegrenzer (STB), Sicherheitsdruckbegrenzer (SDB), Übertemperatur der Warmwasserbereitung (WWB), Sicherheitsventile, Hauptpumpen, Keilriemenwächter, Frequenzumformer, Kälteanlagen, Spannungsausfall usw
// Safety temperature limiter, safety pressure limiter, excess temperature of water heating, safety valves, main pumps, V-belt monitors, frequency converters, refrigeration systems, voltage failure, etc.
AlarmMsg.iParent							:= THIS^;
AlarmMsg.iLabel								:= LblCtl_EvtCategoryAlarmMessage;
AlarmMsg.eDPADMode							:= E_BA_DPADMode.eInclude;																						
AlarmMsg.EC.nInstanceID						:= EC_ID.NC30;
AlarmMsg.EC.iLabel							:= LblFun_ObjectNotificationClass;
AlarmMsg.EC.sObjectName						:= '{Idx=30}'	;
AlarmMsg.EC.eAlarmMode						:= E_BA_AlarmMode.UserDefined;
AlarmMsg.EC.eEventType						:= E_BA_EventType.eAlarm;
AlarmMsg.EC.aPriority[1]					:= 70;
AlarmMsg.EC.aPriority[2]					:= 71;
AlarmMsg.EC.aPriority[3]					:= 72;
AlarmMsg.EC.aAcknowledgeRequired[1]			:= TRUE;
AlarmMsg.EC.aAcknowledgeRequired[2]			:= FALSE;
AlarmMsg.EC.aAcknowledgeRequired[3]			:= TRUE;

//===================================================================
// Ereigniskategorie - Störungsmeldung - Meldung weist auf einen anormalen Betriebszustand hin
// Event category - malfunction message - message indicates abnormal operating condition
// Temperaturwächter (TW), Druckwächter (DW), Temperaturüberwachung von Wärmetauscher (WT) und WWB, Motorschutz, Aufzug-Sammelstörmeldung, Netzdrücke usw.
// Temperature monitor, pressure monitor, temperature monitoring of heat exchanger and water heating, motor protection, lift collective fault signal, mains pressures, etc.
FaultMsg.iParent							:= THIS^;
FaultMsg.iLabel								:= LblCtl_EvtCategoryFaultMessage;
FaultMsg.eDPADMode							:= E_BA_DPADMode.eInclude;																						
FaultMsg.EC.nInstanceID						:= EC_ID.NC40;
FaultMsg.EC.iLabel							:= LblFun_ObjectNotificationClass;
FaultMsg.EC.sObjectName						:= '{Idx=40}'	;
FaultMsg.EC.eAlarmMode						:= E_BA_AlarmMode.UserDefined;
FaultMsg.EC.eEventType						:= E_BA_EventType.eDisturb;
FaultMsg.EC.aPriority[1]					:= 100;
FaultMsg.EC.aPriority[2]					:= 101;
FaultMsg.EC.aPriority[3]					:= 102;
FaultMsg.EC.aAcknowledgeRequired[1]			:= TRUE;
FaultMsg.EC.aAcknowledgeRequired[2]			:= FALSE;
FaultMsg.EC.aAcknowledgeRequired[3]			:= FALSE;
//===================================================================
// Ereigniskategorie - Wartungsmeldung, Hinweis auf Wartungsaktivität o.ä.
// Event category - Maintenance message Maintenance message, indication of maintenance activity or similar.
// Betriebsstunden, Behälterstand, Reparaturschalter usw.
// Operating hours, tank level, repair switch, etc.
MaintenanceMsg01.iParent					:= THIS^;
MaintenanceMsg01.iLabel						:= LblCtl_EvtCategoryMaintenanceMessage;
MaintenanceMsg01.eDPADMode					:= E_BA_DPADMode.eInclude;																						
MaintenanceMsg01.EC.nInstanceID				:= EC_ID.NC50;
MaintenanceMsg01.EC.iLabel					:= LblFun_ObjectNotificationClass;
MaintenanceMsg01.EC.sObjectName				:= '{Idx=50}'	;
MaintenanceMsg01.EC.eAlarmMode				:= E_BA_AlarmMode.UserDefined;
MaintenanceMsg01.EC.eEventType				:= E_BA_EventType.eMaintenance;
MaintenanceMsg01.EC.aPriority[1]			:= 130;
MaintenanceMsg01.EC.aPriority[2]			:= 131;
MaintenanceMsg01.EC.aPriority[3]			:= 132;
MaintenanceMsg01.EC.aAcknowledgeRequired[1]	:= TRUE;
MaintenanceMsg01.EC.aAcknowledgeRequired[2]	:= FALSE;
MaintenanceMsg01.EC.aAcknowledgeRequired[3]	:= FALSE;

// Filterende erreicht, Filter verschmutzt usw.
// Filter end reached, filter dirty, etc.
MaintenanceMsg02.iParent					:= THIS^;
MaintenanceMsg02.iLabel						:= LblCtl_EvtCategoryMaintenanceMessage;
MaintenanceMsg02.eDPADMode					:= E_BA_DPADMode.eInclude;																						
MaintenanceMsg02.EC.nInstanceID				:= EC_ID.NC51;
MaintenanceMsg02.EC.iLabel					:= LblFun_ObjectNotificationClass;
MaintenanceMsg02.EC.sObjectName				:= '{Idx=51}'	;
MaintenanceMsg02.EC.eAlarmMode				:= E_BA_AlarmMode.UserDefined;
MaintenanceMsg02.EC.eEventType				:= E_BA_EventType.eMaintenance;
MaintenanceMsg02.EC.aPriority[1]			:= 135;
MaintenanceMsg02.EC.aPriority[2]			:= 136;
MaintenanceMsg02.EC.aPriority[3]			:= 137;
MaintenanceMsg02.EC.aAcknowledgeRequired[1]	:= TRUE;
MaintenanceMsg02.EC.aAcknowledgeRequired[2]	:= FALSE;
MaintenanceMsg02.EC.aAcknowledgeRequired[3]	:= FALSE;
//===================================================================
//===================================================================
// Ereigniskategorie - Systemmeldung, Störungsmeldung aus GA-System
// Event category - System message, System message, Fault message from building automation system
// Gerätestörung, Batteriemeldung, Kommunikationsunterbrechung usw.
// Unit malfunction, battery message, communication interruption, etc.
SystemMsg.iParent							:= THIS^;
SystemMsg.iLabel							:= LblCtl_EvtCategorySystem;
SystemMsg.eDPADMode							:= E_BA_DPADMode.eInclude;																						
SystemMsg.EC.nInstanceID					:= EC_ID.NC60;
SystemMsg.EC.iLabel							:= LblFun_ObjectNotificationClass;
SystemMsg.EC.sObjectName					:='{Idx=60}';
SystemMsg.EC.eAlarmMode						:= E_BA_AlarmMode.UserDefined;
SystemMsg.EC.eEventType						:= E_BA_EventType.eNotification;
SystemMsg.EC.aPriority[1]					:= 180;
SystemMsg.EC.aPriority[2]					:= 181;
SystemMsg.EC.aPriority[3]					:= 182;
SystemMsg.EC.aAcknowledgeRequired[1]		:= FALSE;
SystemMsg.EC.aAcknowledgeRequired[2]		:= FALSE;
SystemMsg.EC.aAcknowledgeRequired[3]		:= FALSE;
//===================================================================//
//	Ereigniskategorie - Manual operation, Handeingriff
ManualOp.iParent							:= THIS^;
ManualOp.iLabel								:= LblCtl_EvtCategoryManualOperation;
ManualOp.eDPADMode							:= E_BA_DPADMode.eInclude;																						
ManualOp.EC.nInstanceID						:= EC_ID.NC70;
ManualOp.EC.iLabel							:= LblFun_ObjectNotificationClass;
ManualOp.EC.sObjectName						:='{Idx=70}';
ManualOp.EC.eAlarmMode						:= E_BA_AlarmMode.UserDefined;
ManualOp.EC.eEventType						:= E_BA_EventType.eOther;
ManualOp.EC.aPriority[1]					:= 220;
ManualOp.EC.aPriority[2]					:= 220;
ManualOp.EC.aPriority[3]					:= 220;
ManualOp.EC.aAcknowledgeRequired[1]			:= FALSE;
ManualOp.EC.aAcknowledgeRequired[2]			:= FALSE;
ManualOp.EC.aAcknowledgeRequired[3]			:= FALSE;
//===================================================================//
// Ereigniskategorie - Freibleibend, Sonstige Meldungen
// Event category - Other message, Not binding, Other messages
// Betriebszustandswechsel, Betriebsarten, Trendspeicher voll usw.
// Operating status change, operating modes, trend memory full, etc.
OtherMsg.iParent							:= THIS^;
OtherMsg.iLabel								:= LblCtl_EvtCategoryOther;
OtherMsg.eDPADMode							:= E_BA_DPADMode.eInclude;																						
OtherMsg.EC.nInstanceID						:= EC_ID.NC80;
OtherMsg.EC.iLabel							:= LblFun_ObjectNotificationClass;
OtherMsg.EC.sObjectName						:='{Idx=80}';
OtherMsg.EC.eAlarmMode						:= E_BA_AlarmMode.UserDefined;
OtherMsg.EC.eEventType						:= E_BA_EventType.eOther;
OtherMsg.EC.aPriority[1]					:= 230;
OtherMsg.EC.aPriority[2]					:= 231;
OtherMsg.EC.aPriority[3]					:= 232;
OtherMsg.EC.aAcknowledgeRequired[1]			:= FALSE;
OtherMsg.EC.aAcknowledgeRequired[2]			:= FALSE;
OtherMsg.EC.aAcknowledgeRequired[3]			:= FALSE;
END_METHOD

END_FUNCTION_BLOCK

// ---- Templates/POUs/Trade/AutomationControl/EventClasses/FB_BA_EvtGroupsAMEV2017.TcPOU
{region '#Template'}
	{attribute 'Version' := '5.0.0.0'}
	{attribute 'Tags' := '"LCID": "1031", "Text": "General, Cabinet, Control cabinet, Event groups, Categories, Notification classes, Event classes"'}
	{attribute 'Tags' := '"LCID": "1033", "Text": "General, Cabinet, Control cabinet, Event groups, Categories, Notification classes, Event classes"'}
	{attribute 'Using' := '"Type": "Template", "URI": "EC_ID"'}
	{attribute 'Description' := '"LCID": "1031", "Text": "Ereignisgruppen, Kategorien"'}
	{attribute 'Description' := '"LCID": "1033", "Text": "Event groups, categories"'}
{endregion}
FUNCTION_BLOCK FB_BA_EvtGroupsAMEV2017 EXTENDS FB_BA_View
VAR_INPUT CONSTANT
	LifeSafety						: FB_BA_EvtCategory;
	SafetyMsg						: FB_BA_EvtCategory;
	AlarmMsg						: FB_BA_EvtCategory;
	FaultMsg						: FB_BA_EvtCategory;
	MaintenanceMsg01				: FB_BA_EvtCategory;
	MaintenanceMsg02				: FB_BA_EvtCategory;
	SystemMsg						: FB_BA_EvtCategory;
	ManualOp						: FB_BA_EvtCategory;
	OtherMsg						: FB_BA_EvtCategory;
END_VAR

SUPER^(); // FB_BA_View
LifeSafety(); // FB_BA_EvtCategory
SafetyMsg(); // FB_BA_EvtCategory
AlarmMsg(); // FB_BA_EvtCategory
FaultMsg(); // FB_BA_EvtCategory
MaintenanceMsg01(); // FB_BA_EvtCategory
MaintenanceMsg02(); // FB_BA_EvtCategory
SystemMsg(); // FB_BA_EvtCategory
ManualOp(); // FB_BA_EvtCategory
OtherMsg(); // FB_BA_EvtCategory

METHOD FB_init : BOOL
VAR_INPUT
	bInitRetains : BOOL; // if TRUE, the retain variables are initialized (warm start / cold start)
	bInCopyCode : BOOL;  // if TRUE, the instance afterwards gets moved into the copy code (online change)
END_VAR
//===================================================================
// Ereigniskategorie - Gefahr für Leben // Event category - Danger to life
// Brandalarm, Überfall // Fire alarm, robbery
LifeSafety.iParent							:= THIS^;
LifeSafety.iLabel							:= LblCtl_EvtCategoryLifeSafty;
LifeSafety.eDPADMode						:= E_BA_DPADMode.eInclude;																						
LifeSafety.EC.nInstanceID					:= EC_ID.NC10;
LifeSafety.EC.iLabel						:= LblFun_ObjectNotificationClass;
LifeSafety.EC.sObjectName					:='{Idx=10}';
LifeSafety.EC.eAlarmMode					:= E_BA_AlarmMode.eExtended;
LifeSafety.EC.eEventType					:= E_BA_EventType.eAlarm;
LifeSafety.EC.aPriority[1]					:= 10;
LifeSafety.EC.aPriority[2]					:= 11;
LifeSafety.EC.aPriority[3]					:= 12;
//===================================================================		
// Ereigniskategorie - Gefahrenmeldung, Sicherheitsmeldung // Event category - hazard alert, safety message
// Einbruch, unberechtigter Zutritt // Burglary, unauthorised entry
SafetyMsg.iParent							:= THIS^;
SafetyMsg.iLabel							:= LblCtl_EvtCategorySaftyMessage;
SafetyMsg.eDPADMode							:= E_BA_DPADMode.eInclude;																						
SafetyMsg.EC.nInstanceID					:= EC_ID.NC20;
SafetyMsg.EC.iLabel							:= LblFun_ObjectNotificationClass;
SafetyMsg.EC.sObjectName					:='{Idx=20}';
SafetyMsg.EC.eAlarmMode						:= E_BA_AlarmMode.eExtended;
SafetyMsg.EC.eEventType						:= E_BA_EventType.eAlarm;
SafetyMsg.EC.aPriority[1]					:= 40;
SafetyMsg.EC.aPriority[2]					:= 41;
SafetyMsg.EC.aPriority[3]					:= 42;
//===================================================================//
// Ereigniskategorie - Alarmeldung - Meldung signalisiert Anlagenausfall oder erfordert sofortigen Eingriff 
// Event category - Alarm message - Message signals system failure or requires immediate intervention 
// Sicherheitstemperaturbegrenzer (STB), Sicherheitsdruckbegrenzer (SDB), Übertemperatur der Warmwasserbereitung (WWB), Sicherheitsventile, Hauptpumpen, Keilriemenwächter, Frequenzumformer, Kälteanlagen, Spannungsausfall usw
// Safety temperature limiter, safety pressure limiter, excess temperature of water heating, safety valves, main pumps, V-belt monitors, frequency converters, refrigeration systems, voltage failure, etc.
AlarmMsg.iParent							:= THIS^;
AlarmMsg.iLabel								:= LblCtl_EvtCategoryAlarmMessage;
AlarmMsg.eDPADMode							:= E_BA_DPADMode.eInclude;																						
AlarmMsg.EC.nInstanceID						:= EC_ID.NC30;
AlarmMsg.EC.iLabel							:= LblFun_ObjectNotificationClass;
AlarmMsg.EC.sObjectName						:= '{Idx=30}'	;
AlarmMsg.EC.eAlarmMode						:= E_BA_AlarmMode.eExtended;
AlarmMsg.EC.eEventType						:= E_BA_EventType.eAlarm;
AlarmMsg.EC.aPriority[1]					:= 70;
AlarmMsg.EC.aPriority[2]					:= 71;
AlarmMsg.EC.aPriority[3]					:= 72;
//===================================================================
// Ereigniskategorie - Störungsmeldung - Meldung weist auf einen anormalen Betriebszustand hin
// Event category - malfunction message - message indicates abnormal operating condition
// Temperaturwächter (TW), Druckwächter (DW), Temperaturüberwachung von Wärmetauscher (WT) und WWB, Motorschutz, Aufzug-Sammelstörmeldung, Netzdrücke usw.
// Temperature monitor, pressure monitor, temperature monitoring of heat exchanger and water heating, motor protection, lift collective fault signal, mains pressures, etc.
FaultMsg.iParent							:= THIS^;
FaultMsg.iLabel								:= LblCtl_EvtCategoryFaultMessage;
FaultMsg.eDPADMode							:= E_BA_DPADMode.eInclude;																						
FaultMsg.EC.nInstanceID						:= EC_ID.NC40;
FaultMsg.EC.iLabel							:= LblFun_ObjectNotificationClass;
FaultMsg.EC.sObjectName						:= '{Idx=40}'	;
FaultMsg.EC.eAlarmMode						:= E_BA_AlarmMode.eStandard;
FaultMsg.EC.eEventType						:= E_BA_EventType.eDisturb;
FaultMsg.EC.aPriority[1]					:= 100;
FaultMsg.EC.aPriority[2]					:= 101;
FaultMsg.EC.aPriority[3]					:= 102;
//===================================================================
// Ereigniskategorie - Wartungsmeldung, Hinweis auf Wartungsaktivität o.ä.
// Event category - Maintenance message Maintenance message, indication of maintenance activity or similar.
// Betriebsstunden, Behälterstand, Reparaturschalter usw.
// Operating hours, tank level, repair switch, etc.
MaintenanceMsg01.iParent					:= THIS^;
MaintenanceMsg01.iLabel						:= LblCtl_EvtCategoryMaintenanceMessage;
MaintenanceMsg01.eDPADMode					:= E_BA_DPADMode.eInclude;																						
MaintenanceMsg01.EC.nInstanceID				:= EC_ID.NC50;
MaintenanceMsg01.EC.iLabel					:= LblFun_ObjectNotificationClass;
MaintenanceMsg01.EC.sObjectName				:= '{Idx=50}'	;
MaintenanceMsg01.EC.eAlarmMode				:= E_BA_AlarmMode.eStandard;
MaintenanceMsg01.EC.eEventType				:= E_BA_EventType.eMaintenance;
MaintenanceMsg01.EC.aPriority[1]			:= 130;
MaintenanceMsg01.EC.aPriority[2]			:= 131;
MaintenanceMsg01.EC.aPriority[3]			:= 132;
// Filterende erreicht, Filter verschmutzt usw.
// Filter end reached, filter dirty, etc.
MaintenanceMsg02.iParent					:= THIS^;
MaintenanceMsg02.iLabel						:= LblCtl_EvtCategoryMaintenanceMessage;
MaintenanceMsg02.eDPADMode					:= E_BA_DPADMode.eInclude;																						
MaintenanceMsg02.EC.nInstanceID				:= EC_ID.NC51;
MaintenanceMsg02.EC.iLabel					:= LblFun_ObjectNotificationClass;
MaintenanceMsg02.EC.sObjectName				:= '{Idx=51}'	;
MaintenanceMsg02.EC.eAlarmMode				:= E_BA_AlarmMode.eStandard;
MaintenanceMsg02.EC.eEventType				:= E_BA_EventType.eMaintenance;
MaintenanceMsg02.EC.aPriority[1]			:= 135;
MaintenanceMsg02.EC.aPriority[2]			:= 136;
MaintenanceMsg02.EC.aPriority[3]			:= 137;
//===================================================================
//===================================================================
// Ereigniskategorie - Systemmeldung, Störungsmeldung aus GA-System
// Event category - System message, System message, Fault message from building automation system
// Gerätestörung, Batteriemeldung, Kommunikationsunterbrechung usw.
// Unit malfunction, battery message, communication interruption, etc.
SystemMsg.iParent							:= THIS^;
SystemMsg.iLabel							:= LblCtl_EvtCategorySystem;
SystemMsg.eDPADMode							:= E_BA_DPADMode.eInclude;																						
SystemMsg.EC.nInstanceID					:= EC_ID.NC60;
SystemMsg.EC.iLabel							:= LblFun_ObjectNotificationClass;
SystemMsg.EC.sObjectName					:='{Idx=60}';
SystemMsg.EC.eAlarmMode						:= E_BA_AlarmMode.eSimple;
SystemMsg.EC.eEventType						:= E_BA_EventType.eNotification;
SystemMsg.EC.aPriority[1]					:= 180;
SystemMsg.EC.aPriority[2]					:= 181;
SystemMsg.EC.aPriority[3]					:= 182;
//===================================================================//
//	Ereigniskategorie - Manual operation, Handeingriff
ManualOp.iParent							:= THIS^;
ManualOp.iLabel								:= LblCtl_EvtCategoryManualOperation;
ManualOp.eDPADMode							:= E_BA_DPADMode.eInclude;																						
ManualOp.EC.nInstanceID						:= EC_ID.NC70;
ManualOp.EC.iLabel							:= LblFun_ObjectNotificationClass;
ManualOp.EC.sObjectName						:='{Idx=70}';
ManualOp.EC.eAlarmMode						:= E_BA_AlarmMode.eSimple;
ManualOp.EC.eEventType						:= E_BA_EventType.eOther;
ManualOp.EC.aPriority[1]					:= 220;
ManualOp.EC.aPriority[2]					:= 220;
ManualOp.EC.aPriority[3]					:= 220;
//===================================================================//
// Ereigniskategorie - Freibleibend, Sonstige Meldungen
// Event category - Other message, Not binding, Other messages
// Betriebszustandswechsel, Betriebsarten, Trendspeicher voll usw.
// Operating status change, operating modes, trend memory full, etc.
OtherMsg.iParent							:= THIS^;
OtherMsg.iLabel								:= LblCtl_EvtCategoryOther;
OtherMsg.eDPADMode							:= E_BA_DPADMode.eInclude;																						
OtherMsg.EC.nInstanceID						:= EC_ID.NC80;
OtherMsg.EC.iLabel							:= LblFun_ObjectNotificationClass;
OtherMsg.EC.sObjectName						:='{Idx=80}';
OtherMsg.EC.eAlarmMode						:= E_BA_AlarmMode.eSimple;
OtherMsg.EC.eEventType						:= E_BA_EventType.eOther;
OtherMsg.EC.aPriority[1]					:= 230;
OtherMsg.EC.aPriority[2]					:= 231;
OtherMsg.EC.aPriority[3]					:= 232;
END_METHOD

END_FUNCTION_BLOCK

// ---- Templates/POUs/Trade/BuildingAutomation/General/FB_BA_BuildingData.TcPOU
{region '#Template'}
	{attribute 'Version' := '5.1.0.0'}
	{attribute 'Tags' := '"LCID": "1031", "Text": "Gewerk, Gebäudeautomation, Daten"'}
	{attribute 'Tags' := '"LCID": "1033", "Text": "Trade, Building automation, data"'}
	{attribute 'Using' := '"Type": "Template", "URI": "Site"'}
	{attribute 'Description' := '"LCID": "1031", "Text": "Aufruf der Aggregate der allgemeinen Gebäudedaten"'}
	{attribute 'Description' := '"LCID": "1033", "Text": "Calling the aggrgates of common building data"'}
{endregion}	 
FUNCTION_BLOCK FB_BA_BuildingData EXTENDS FB_BA_View
VAR_INPUT
END_VAR
VAR_OUTPUT
END_VAR
VAR_INPUT CONSTANT
	BuildingEnergLvl			: FB_BA_BuildingEnergyLevel;
	BuildingSpRmT				: FB_BA_BuildingSpRmT;
END_VAR
VAR
END_VAR

SUPER^(); // FB_BA_View
BuildingEnergLvl(); // FB_BA_BuildingEnergyLevel
BuildingSpRmT(); // FB_BA_BuildingSpRmT

METHOD FB_init : BOOL
VAR_INPUT
	bInitRetains : BOOL; // if TRUE, the retain variables are initialized (warm start / cold start)
	bInCopyCode : BOOL;  // if TRUE, the instance afterwards gets moved into the copy code (online change)
END_VAR
BuildingEnergLvl.iParent		:= THIS^;	
BuildingEnergLvl.iLabel			:= LblCtl_BuildingEnergyLevel;  
BuildingEnergLvl.sObjectName	:= '{Idx=01}';
BuildingEnergLvl.eDPADMode		:= E_BA_DPADMode.eInclude;

BuildingSpRmT.iParent			:= THIS^;	
BuildingSpRmT.iLabel			:= LblCtl_BuildingSpRmT;  
BuildingSpRmT.sObjectName		:= '{Idx=02}';
BuildingSpRmT.eDPADMode			:= E_BA_DPADMode.eInclude;
END_METHOD

END_FUNCTION_BLOCK

// ---- Templates/POUs/Trade/HeatingSystem/General/FB_BA_H_OpMod.TcPOU
{region '#Template'}
	{attribute 'Version' := '5.0.0.0'}
	{attribute 'Tags' := '"LCID": "1031", "Text": "H, General, HtgCir, Operating mode"'}
	{attribute 'Tags' := '"LCID": "1033", "Text": "H, General, HtgCir, Operating mode"'}
	{attribute 'Using' := '"Type": "Template", "URI": "E_BA_OnOff"'}
	{attribute 'Using' := '"Type": "Template", "URI": "E_BA_EnergyLvl"'}		 
	{attribute 'Using' := '"Type": "Template", "URI": "E_BA_EnergyLvlA"'}		 
	{attribute 'Description' := '"LCID": "1031", "Text": "Betriebsart"'}
	{attribute 'Description' := '"LCID": "1033", "Text": "Operating mode"'}
{endregion}
FUNCTION_BLOCK FB_BA_H_OpMod EXTENDS FB_BA_View
VAR_INPUT
	bDst					: BOOL;
	bHtgLmt					: BOOL;
	bTWthLowLimit			: BOOL;
END_VAR
VAR_OUTPUT
	eOpMod					: E_BA_EnergyLvl;
	bRls					: BOOL;
END_VAR
VAR_INPUT CONSTANT
	OpModMan				: FB_BA_MV_Op;
	Sched					: FB_BA_SchedM;
	OpModPr					: FB_BA_MV_Op;								 
	Rls						: FB_BA_BV_Op;
END_VAR
VAR
	OpModSwi				: FB_BA_PrioSwi_UDI08;
	RlsMMux					: FB_BA_MMUX_B04;
END_VAR

SUPER^(); // FB_BA_View
OpModMan(); // FB_BA_MV_Op
Sched(); // FB_BA_SchedM
OpModSwi(
    bEn01 := bDst,
    nVal01 := E_BA_EnergyLvl.eProtection,
    bEn02 := OpModMan.nPresentValue = E_BA_EnergyLvlA.eProtection,
    nVal02 := E_BA_EnergyLvl.eProtection,
    bEn03 := OpModMan.nPresentValue = E_BA_EnergyLvlA.eEconomy,
    nVal03 := E_BA_EnergyLvl.eEconomy,
    bEn04 := OpModMan.nPresentValue = E_BA_EnergyLvlA.eComfort,
    nVal04 := E_BA_EnergyLvl.eComfort,
    bEn05 := NOT bHtgLmt,
    nVal05 := E_BA_EnergyLvl.eProtection,
    bEn06 := Sched.nPresentValue = E_BA_EnergyLvl.eProtection,
    nVal06 := E_BA_EnergyLvl.eProtection,
    bEn07 := Sched.nPresentValue = E_BA_EnergyLvl.eEconomy,
    nVal07 := E_BA_EnergyLvl.eEconomy,
    bEn08 := Sched.nPresentValue = E_BA_EnergyLvl.eComfort,
    nVal08 := E_BA_EnergyLvl.eComfort); // FB_BA_PrioSwi_UDI08
OpModPr(nValuePgm := OpModSwi.nVal); // FB_BA_MV_Op
eOpMod := OpModPr.nPresentValue;
RlsMMux(
    bEn := TRUE,
    nSel := eOpMod,
    nEn01 := E_BA_EnergyLvl.eProtection,
    bVal01 := bTWthLowLimit,
    nEn02 := E_BA_EnergyLvl.eEconomy,
    bVal02 := TRUE,
    nEn03 := E_BA_EnergyLvl.eComfort,
    bVal03 := TRUE); // FB_BA_MMUX_B04
Rls(bValuePgm := RlsMMux.bVal); // FB_BA_BV_Op
bRls := Rls.bPresentValue;

METHOD FB_init : BOOL
VAR_INPUT
	bInitRetains : BOOL; // if TRUE, the retain variables are initialized (warm start / cold start)
	bInCopyCode : BOOL;  // if TRUE, the instance afterwards gets moved into the copy code (online change)
END_VAR
OpModMan.iParent										:= THIS^;
OpModMan.iLabel											:= LblCtl_OperationModeSelection; 
OpModMan.aStateText[1]									:= txtEvent_Auto;
OpModMan.aStateText[2]									:= txtEvent_Protection;
OpModMan.aStateText[3]									:= txtEvent_Economy;
OpModMan.aStateText[4]									:= txtEvent_Comfort;
OpModMan.nValueRm										:= 1;
                        								
OpModPr.iParent											:= THIS^;
OpModPr.iLabel											:= LblCtl_PresentOperationMode; 
OpModPr.aStateText[1]									:= txtEvent_Protection; 
OpModPr.aStateText[2]									:= txtEvent_Economy; 
OpModPr.aStateText[3]									:= txtEvent_Comfort; 
OpModPr.nValueRm										:= 1;
                        								
Rls.iParent												:= THIS^;
Rls.iLabel												:= LblFun_Enabled; 
Rls.sInactiveText										:= txtEvent_Off;
Rls.sActiveText											:= txtEvent_On;	
Rls.bValueRm											:= FALSE;								
Rls.eToggleMode 										:= E_BA_ToggleMode.eSwitch;	
                        	
Sched.iParent											:= THIS^;
Sched.iLabel											:= LblFun_Scheduler; 
Sched.aStateText[1]										:= txtEvent_Protection;
Sched.aStateText[2]										:= txtEvent_Economy;
Sched.aStateText[3]										:= txtEvent_Comfort;
Sched.nPredictTime										:= 0;
Sched.nDefaultValue										:= E_BA_EnergyLvl.eProtection;
Sched.bWriteWeekly										:= FALSE;
//	Monday
Sched.aWeek[E_BA_Weekday.eMonday,1].eState				:= E_BA_SchedEntryState.eValue;
Sched.aWeek[E_BA_Weekday.eMonday,1].uValue.udiVal		:= E_BA_EnergyLvl.eComfort;
Sched.aWeek[E_BA_Weekday.eMonday,1].stTime.nHour		:= 6;
Sched.aWeek[E_BA_Weekday.eMonday,1].stTime.nMinute		:= 0;
Sched.aWeek[E_BA_Weekday.eMonday,1].stTime.nSecond		:= 0;
Sched.aWeek[E_BA_Weekday.eMonday,2].eState				:= E_BA_SchedEntryState.eValue;
Sched.aWeek[E_BA_Weekday.eMonday,2].uValue.udiVal		:= E_BA_EnergyLvl.eEconomy;
Sched.aWeek[E_BA_Weekday.eMonday,2].stTime.nHour		:= 20;
Sched.aWeek[E_BA_Weekday.eMonday,2].stTime.nMinute		:= 0;
Sched.aWeek[E_BA_Weekday.eMonday,2].stTime.nSecond		:= 0;
Sched.aWeek[E_BA_Weekday.eMonday,3].eState				:= E_BA_SchedEntryState.eValue;
Sched.aWeek[E_BA_Weekday.eMonday,3].uValue.udiVal		:= E_BA_EnergyLvl.eProtection;
Sched.aWeek[E_BA_Weekday.eMonday,3].stTime.nHour		:= 0;
Sched.aWeek[E_BA_Weekday.eMonday,3].stTime.nMinute		:= 0;
Sched.aWeek[E_BA_Weekday.eMonday,3].stTime.nSecond		:= 0;
//	Tuesday
Sched.aWeek[E_BA_Weekday.eTuesday,1].eState				:= E_BA_SchedEntryState.eValue;
Sched.aWeek[E_BA_Weekday.eTuesday,1].uValue.udiVal		:= E_BA_EnergyLvl.eComfort;
Sched.aWeek[E_BA_Weekday.eTuesday,1].stTime.nHour		:= 6;
Sched.aWeek[E_BA_Weekday.eTuesday,1].stTime.nMinute		:= 0;
Sched.aWeek[E_BA_Weekday.eTuesday,1].stTime.nSecond		:= 0;
Sched.aWeek[E_BA_Weekday.eTuesday,2].eState				:= E_BA_SchedEntryState.eValue;
Sched.aWeek[E_BA_Weekday.eTuesday,2].uValue.udiVal		:= E_BA_EnergyLvl.eEconomy;
Sched.aWeek[E_BA_Weekday.eTuesday,2].stTime.nHour		:= 20;
Sched.aWeek[E_BA_Weekday.eTuesday,2].stTime.nMinute		:= 0;
Sched.aWeek[E_BA_Weekday.eTuesday,2].stTime.nSecond		:= 0;
Sched.aWeek[E_BA_Weekday.eTuesday,3].eState				:= E_BA_SchedEntryState.eValue;
Sched.aWeek[E_BA_Weekday.eTuesday,3].uValue.udiVal		:= E_BA_EnergyLvl.eProtection;
Sched.aWeek[E_BA_Weekday.eTuesday,3].stTime.nHour		:= 0;
Sched.aWeek[E_BA_Weekday.eTuesday,3].stTime.nMinute		:= 0;
Sched.aWeek[E_BA_Weekday.eTuesday,3].stTime.nSecond		:= 0;
//	Wednesday
Sched.aWeek[E_BA_Weekday.eWednesday,1].eState			:= E_BA_SchedEntryState.eValue;
Sched.aWeek[E_BA_Weekday.eWednesday,1].uValue.udiVal	:= E_BA_EnergyLvl.eComfort;
Sched.aWeek[E_BA_Weekday.eWednesday,1].stTime.nHour		:= 6;
Sched.aWeek[E_BA_Weekday.eWednesday,1].stTime.nMinute	:= 0;
Sched.aWeek[E_BA_Weekday.eWednesday,1].stTime.nSecond	:= 0;
Sched.aWeek[E_BA_Weekday.eWednesday,2].eState			:= E_BA_SchedEntryState.eValue;
Sched.aWeek[E_BA_Weekday.eWednesday,2].uValue.udiVal	:= E_BA_EnergyLvl.eEconomy;
Sched.aWeek[E_BA_Weekday.eWednesday,2].stTime.nHour		:= 20;
Sched.aWeek[E_BA_Weekday.eWednesday,2].stTime.nMinute	:= 0;
Sched.aWeek[E_BA_Weekday.eWednesday,2].stTime.nSecond	:= 0;
Sched.aWeek[E_BA_Weekday.eWednesday,3].eState			:= E_BA_SchedEntryState.eValue;
Sched.aWeek[E_BA_Weekday.eWednesday,3].uValue.udiVal	:= E_BA_EnergyLvl.eProtection;
Sched.aWeek[E_BA_Weekday.eWednesday,3].stTime.nHour		:= 0;
Sched.aWeek[E_BA_Weekday.eWednesday,3].stTime.nMinute	:= 0;
Sched.aWeek[E_BA_Weekday.eWednesday,3].stTime.nSecond	:= 0;
//	Thursday
Sched.aWeek[E_BA_Weekday.eThursday,1].eState			:= E_BA_SchedEntryState.eValue;
Sched.aWeek[E_BA_Weekday.eThursday,1].uValue.udiVal		:=E_BA_EnergyLvl.eComfort;
Sched.aWeek[E_BA_Weekday.eThursday,1].stTime.nHour		:= 6;
Sched.aWeek[E_BA_Weekday.eThursday,1].stTime.nMinute	:= 0;
Sched.aWeek[E_BA_Weekday.eThursday,1].stTime.nSecond	:= 0;
Sched.aWeek[E_BA_Weekday.eThursday,2].eState			:= E_BA_SchedEntryState.eValue;
Sched.aWeek[E_BA_Weekday.eThursday,2].uValue.udiVal		:= E_BA_EnergyLvl.eEconomy;
Sched.aWeek[E_BA_Weekday.eThursday,2].stTime.nHour		:= 20;
Sched.aWeek[E_BA_Weekday.eThursday,2].stTime.nMinute	:= 0;
Sched.aWeek[E_BA_Weekday.eThursday,2].stTime.nSecond	:= 0;
Sched.aWeek[E_BA_Weekday.eThursday,3].eState			:= E_BA_SchedEntryState.eValue;
Sched.aWeek[E_BA_Weekday.eThursday,3].uValue.udiVal		:= E_BA_EnergyLvl.eProtection;
Sched.aWeek[E_BA_Weekday.eThursday,3].stTime.nHour		:= 0;
Sched.aWeek[E_BA_Weekday.eThursday,3].stTime.nMinute	:= 0;
Sched.aWeek[E_BA_Weekday.eThursday,3].stTime.nSecond	:= 0;
//	Friday
Sched.aWeek[E_BA_Weekday.eFriday,1].eState				:= E_BA_SchedEntryState.eValue;
Sched.aWeek[E_BA_Weekday.eFriday,1].uValue.udiVal		:= E_BA_EnergyLvl.eComfort;
Sched.aWeek[E_BA_Weekday.eFriday,1].stTime.nHour		:= 6;
Sched.aWeek[E_BA_Weekday.eFriday,1].stTime.nMinute		:= 0;
Sched.aWeek[E_BA_Weekday.eFriday,1].stTime.nSecond		:= 0;
Sched.aWeek[E_BA_Weekday.eFriday,2].eState				:= E_BA_SchedEntryState.eValue;
Sched.aWeek[E_BA_Weekday.eFriday,2].uValue.udiVal		:= E_BA_EnergyLvl.eEconomy;
Sched.aWeek[E_BA_Weekday.eFriday,2].stTime.nHour		:= 20;
Sched.aWeek[E_BA_Weekday.eFriday,2].stTime.nMinute		:= 0;
Sched.aWeek[E_BA_Weekday.eFriday,2].stTime.nSecond		:= 0;
Sched.aWeek[E_BA_Weekday.eFriday,3].eState				:= E_BA_SchedEntryState.eValue;
Sched.aWeek[E_BA_Weekday.eFriday,3].uValue.udiVal		:= E_BA_EnergyLvl.eProtection;
Sched.aWeek[E_BA_Weekday.eFriday,3].stTime.nHour		:= 0;
Sched.aWeek[E_BA_Weekday.eFriday,3].stTime.nMinute		:= 0;
Sched.aWeek[E_BA_Weekday.eFriday,3].stTime.nSecond		:= 0;
END_METHOD

END_FUNCTION_BLOCK

// ---- Templates/POUs/Trade/RoomAutomation/Common/DALI FunctionBlocks/FB_BA_LightActrDALI_Base.TcPOU
{region '#Template'}
	{attribute 'Version' := '5.0.0.0'}
	{attribute 'Tags' := '"LCID": "1031", "Text": "RA, Allgemein, DALI, Lichtfaktor"'}
	{attribute 'Tags' := '"LCID": "1033", "Text": "RA, Common, DALI, light-actuator"'}
	{attribute 'Description' := '"LCID": "1031", "Text": "Grundbaustein DALI Lichtaktor"'}
	{attribute 'Description' := '"LCID": "1033", "Text": "Basic function DALI light-actuator"'}
{endregion}
FUNCTION_BLOCK FB_BA_LightActrDALI_Base
VAR_INPUT
	bEn							: BOOL;							// FB-enable
	bInitialize					: BOOL;							// initialize with DALI-parameters
	stLightingCmd				: ST_BA_Lighting;				// command-telegram
	eAdrType					: Tc3_DALI.E_DALIAddressType	:= Tc3_DALI.E_DALIAddressType.Short;
	nAdr						: BYTE;
	nAdrRefDev					: BYTE;							// reference device if group-mode is selected
	ipDALICommunication			: Tc3_DALI.I_DALICommunication;
END_VAR
VAR_OUTPUT
	nActlLgtVal					: BYTE;							// 0..254
	fActlLgtVal					: REAL;							// 0..100
	bInitializing				: BOOL;							// device is being initialized
	bErr						: BOOL;							// error
END_VAR
VAR_INPUT CONSTANT PERSISTENT
{region 'Application parameters'}		
	{attribute 'parameterUnit':= 'DALI'}
	nHysLgtVal					: BYTE;							// hysteresis to accept a new light-value-command
	{attribute 'parameterUnit':= 's'}
	nPrdQueryLgtVal				: UDINT;						// background query light-level
	{attribute 'parameterUnit':= 's'}
	nPrdQueryLgtVal_Fast		: UDINT	:= 10;					// background query light-level fast -> only in case of error to recover more quickly
{endregion}	
	 
{region 'Device parameters to be initially set into the device'}	
	{attribute 'parameterUnit':= 'DALI'}
	nMinLevel					: BYTE	:= 126;					// 1..254
	{attribute 'parameterUnit':= 'DALI'}
	nMaxLevel					: BYTE	:= 254;					// 1..254
	{attribute 'parameterUnit':= 'DALI'}
	nPowerOnLevel				: BYTE	:= 254;					// 1..254
	{attribute 'parameterUnit':= 'DALI'}
	nSystemFailureLevel			: BYTE	:= 254;					// 1..254
	eFadeTime					: Tc3_DALI.E_DALIFadeTime	:= Tc3_DALI.E_DALIFadeTime.Disabled;
	eFadeRate					: Tc3_DALI.E_DALIFadeRate	:= Tc3_DALI.E_DALIFadeRate.N358StepsPerSec;
{endregion}                                                     
END_VAR
VAR CONSTANT
	eExtendedFadeTimeBase		: Tc3_DALI.E_DALIExtendedFadeTimeBase		:= Tc3_DALI.E_DALIExtendedFadeTimeBase.Base01;
	eExtendedFadeTimeMultiplier	: Tc3_DALI.E_DALIExtendedFadeTimeMultiplier	:= Tc3_DALI.E_DALIExtendedFadeTimeMultiplier.Disabled;
END_VAR
VAR
	rtInitialize				: R_TRIG;    
	bInitializationDone			: BOOL	:= TRUE;
	bInitializationErr			: BOOL;
	sInitializationMessage		: T_MaxString;
	
	bSetLightValBusy			: BOOL;
	bSetLightValErr				: BOOL;
	bGetLightValBusy			: BOOL;
	bGetLightValErr				: BOOL;
	
	bInhibit					: BOOL; // Inhibit in case of error
	
	fbLogMsgShortAdr			: FB_BA_LogMessage;
	fbLogMsgGroupAdr			: FB_BA_LogMessage;
	fbLogMsgReferenceDev		: FB_BA_LogMessage;
	fbLogMsgAddresstype			: FB_BA_LogMessage;
	fbLogMsgInterface			: FB_BA_LogMessage;
	fbLogMsgReferenceDevice		: FB_BA_LogMessage;
	
	fbLogMsSetLightValCmdErr	: FB_BA_LogMessage;
	fbLogMsgGetLightValCmdErr	: FB_BA_LogMessage;
	fbLogMsgInitializationErr	: FB_BA_LogMessage;
END_VAR

{region 'errorhandling'}
bErr	:= FALSE;

IF	(nAdr > 63) THEN
	fbLogMsgShortAdr.Show(ADSLOG_MSGTYPE_ERROR, 'DALI addressing error', 'short-address must not exceed 63', FALSE); 	
	bErr	:= TRUE;
	RETURN;
ELSE
	fbLogMsgShortAdr.Reset();	
	bErr	:= FALSE;
END_IF
	 
IF	(eAdrType = Tc3_DALI.E_DALIAddressType.Group) AND_THEN (nAdr > 15) THEN
	fbLogMsgGroupAdr.Show(ADSLOG_MSGTYPE_ERROR, 'DALI addressing error', 'group-Address must not exceed 15', FALSE); 	
	bErr	:= TRUE;
	RETURN;
ELSE
	fbLogMsgGroupAdr.Reset();	
	bErr	:= FALSE;	
END_IF	
	 
IF	((eAdrType = Tc3_DALI.E_DALIAddressType.Group) OR_ELSE (eAdrType = Tc3_DALI.E_DALIAddressType.Broadcast)) AND_THEN (nAdrRefDev > 63) THEN
	fbLogMsgReferenceDev.Show(ADSLOG_MSGTYPE_ERROR, 'DALI addressing error', 'address of reference-device must not exceed 63', FALSE); 	
	bErr	:= TRUE;
	RETURN;
ELSE
	fbLogMsgReferenceDev.Reset();	
	bErr	:= FALSE;	
END_IF	

IF	(eAdrType <> Tc3_DALI.E_DALIAddressType.Short) AND_THEN (eAdrType <> Tc3_DALI.E_DALIAddressType.Group) AND_THEN (eAdrType <> Tc3_DALI.E_DALIAddressType.Broadcast) THEN
	fbLogMsgAddresstype.Show(ADSLOG_MSGTYPE_ERROR, 'DALI addressing error', 'only address-type short, group or broadcast is allowed', FALSE); 	
	bErr	:= TRUE;
	RETURN;
ELSE
	fbLogMsgAddresstype.Reset();	
	bErr	:= FALSE;	
END_IF	
	 
IF	(ipDALICommunication = 0) THEN
	fbLogMsgInterface.Show(ADSLOG_MSGTYPE_ERROR, 'DALI addressing error', 'communication interface-pointer must not be 0', FALSE); 	
	bErr	:= TRUE;
	RETURN;
ELSE
	fbLogMsgInterface.Reset();	
	bErr	:= FALSE;
END_IF	 
{endregion}

{region 'initialization'}
rtInitialize(CLK:=bInitialize);
IF rtInitialize.Q	THEN
	bInitializationDone	:= FALSE;
END_IF

THIS^._Initialization(bStart:= rtInitialize.Q);
IF	bInitializationErr THEN
	CASE eAdrType	OF
		Tc3_DALI.E_DALIAddressType.Short:
			sInitializationMessage:= CONCAT('Single-device #', TO_STRING(nAdr));
		Tc3_DALI.E_DALIAddressType.Group:
			sInitializationMessage:= CONCAT('Group #', TO_STRING(nAdr));	
		Tc3_DALI.E_DALIAddressType.Broadcast:
			sInitializationMessage:= 'Broadcast';
	END_CASE
	sInitializationMessage	:= CONCAT(CONCAT(sInitializationMessage, ','), GetLineInfo());
	fbLogMsgInitializationErr.Show(ADSLOG_MSGTYPE_ERROR, 'DALI initialization-error', sInitializationMessage, FALSE); 	
				   
	bErr	:= TRUE;
	RETURN;
ELSE
	fbLogMsgInitializationErr.Reset();	
	bErr	:= FALSE;
END_IF
{endregion}


THIS^._Execution();

{attribute 'hide'}
METHOD PROTECTED _Execution : BOOL
VAR_INPUT
END_VAR

{region 'Wait to be enabled and initialized'}
IF NOT bEn OR NOT bInitializationDone THEN
	SetLightVal	(bEn	:= FALSE,
				fLgtVal	:= 0); 
	GetLightVal	(bEn	:= FALSE); 
	RETURN;
END_IF
{endregion}

IF eAdrType = Tc3_DALI.E_DALIAddressType.Short	THEN
	nAdrRefDev	:= nAdr;
END_IF

{region 'check group membership of reference-device'}
CheckGroupRefDev	(bEn		:= (eAdrType = Tc3_DALI.E_DALIAddressType.Group));
{endregion}

{region 'set light level'}
SetLightVal	(bEn				:= NOT bInhibit,
			fLgtVal				:= stLightingCmd.fLgtVal); 
{endregion}
	 
{region 'query light level'}	 
GetLightVal	(bEn				:= (nPrdQueryLgtVal>0));
{endregion}

IF bGetLightValErr	THEN	 // GetLightValErr as an indicator, that the device is not defective. If defective, setting Light value and -temperature and polling temperature is not wanted.
	bInhibit:= TRUE;
END_IF
IF NOT bGetLightValBusy	AND NOT bGetLightValErr THEN 
	bInhibit:= FALSE;
END_IF
	 
IF bSetLightValErr	OR bGetLightValErr	THEN
	bErr	:= TRUE;
ELSE
	bErr	:= FALSE;
END_IF
END_METHOD

{attribute 'hide'}
METHOD PROTECTED _Initialization : BOOL
VAR_INPUT
	bStart		: BOOL;
END_VAR

VAR_INST
	
	fbStartQuiescentMode				: FB_DALI103StartQuiescentMode(0);
	fbSetMinLevel						: FB_DALI102SetMinLevel(0);
	fbSetMaxLevel                       : FB_DALI102SetMaxLevel(0);
	fbSetPowerOnLevel					: FB_DALI102SetPowerOnLevel(0);
	fbSetSystemFailureLevel				: FB_DALI102SetSystemFailureLevel(0);
	fbSetFadeTime                       : FB_DALI102SetFadeTime(0);
	fbSetExtendedFadeTime               : FB_DALI102SetExtendedFadeTime(0);
	fbSetFadeRate                       : FB_DALI102SetFadeRate(0);
	fbStopQuiescentMode					: FB_DALI103StopQuiescentMode(0);
			
	nStep								: INT;
	rtStart								: R_TRIG;
END_VAR
fbStartQuiescentMode.ipDALICommunication			:= ipDALICommunication;
fbStartQuiescentMode.nAddress						:= nAdr;

fbSetMinLevel.ipDALICommunication					:= ipDALICommunication;
fbSetMinLevel.nAddress								:= nAdr;
fbSetMinLevel.eAddressType							:= eAdrType;
fbSetMinLevel.nMinLevel								:= nMinLevel;

fbSetMaxLevel.ipDALICommunication					:= ipDALICommunication;
fbSetMaxLevel.nAddress								:= nAdr;
fbSetMaxLevel.eAddressType							:= eAdrType;
fbSetMaxLevel.nMaxLevel								:= nMaxLevel;

fbSetPowerOnLevel.ipDALICommunication				:= ipDALICommunication;
fbSetPowerOnLevel.nAddress							:= nAdr;
fbSetPowerOnLevel.eAddressType						:= eAdrType;
fbSetPowerOnLevel.nPowerOnLevel						:= nPowerOnLevel;

fbSetSystemFailureLevel.ipDALICommunication			:= ipDALICommunication;
fbSetSystemFailureLevel.nAddress					:= nAdr;
fbSetSystemFailureLevel.eAddressType				:= eAdrType;
fbSetSystemFailureLevel.nSystemFailureLevel			:= nSystemFailureLevel;

fbSetFadeTime.ipDALICommunication					:= ipDALICommunication;
fbSetFadeTime.nAddress								:= nAdr;
fbSetFadeTime.eAddressType							:= eAdrType;
fbSetFadeTime.eFadeTime								:= eFadeTime;

fbSetExtendedFadeTime.ipDALICommunication			:= ipDALICommunication;
fbSetExtendedFadeTime.nAddress						:= nAdr;
fbSetExtendedFadeTime.eAddressType					:= eAdrType;
fbSetExtendedFadeTime.eExtendedFadeTimeBase			:= E_DALIExtendedFadeTimeBase.Base01;
fbSetExtendedFadeTime.eExtendedFadeTimeMultiplier	:= E_DALIExtendedFadeTimeMultiplier.Disabled;

fbSetFadeRate.ipDALICommunication					:= ipDALICommunication;
fbSetFadeRate.nAddress								:= nAdr;
fbSetFadeRate.eAddressType							:= eAdrType;
fbSetFadeRate.eFadeRate								:= eFadeRate;

fbStopQuiescentMode.ipDALICommunication				:= ipDALICommunication;
fbStopQuiescentMode.nAddress						:= nAdr;


rtStart(CLK	:= bStart);
IF rtStart.Q	THEN
	bInitializationDone				:= FALSE;
	bInitializationErr				:= FALSE;
	fbStartQuiescentMode			(bStart:=FALSE);
	fbSetMinLevel					(bStart:=FALSE);
	fbSetMaxLevel					(bStart:=FALSE);
	fbSetFadeTime					(bStart:=FALSE);
	fbSetExtendedFadeTime			(bStart:=FALSE);
	fbSetFadeRate					(bStart:=FALSE);
	fbStopQuiescentMode				(bStart:=FALSE);
	
	nStep	:= 10;
END_IF

CASE nStep OF
	0	: 	// Idle
	
	10	:	fbStartQuiescentMode(bStart:=TRUE);
			IF NOT fbStartQuiescentMode.bBusy	THEN
				IF fbStartQuiescentMode.bError	THEN
					nStep	:= 900;
				ELSE	
					nStep	:= 20;
				END_IF
			END_IF
	
	20	:	fbSetMinLevel(bStart:=TRUE);
			IF NOT fbSetMinLevel.bBusy	THEN
				IF fbSetMinLevel.bError	THEN
					nStep	:= 900;
				ELSE	
					nStep	:= 30;
				END_IF
			END_IF
		
	30	:	fbSetMaxLevel(bStart:=TRUE);
			IF NOT fbSetMaxLevel.bBusy	THEN
				IF fbSetMaxLevel.bError	THEN
					nStep	:= 900;
				ELSE	
					nStep	:= 40;
				END_IF
			END_IF
		
	40	:	fbSetPowerOnLevel(bStart:=TRUE);
			IF NOT fbSetPowerOnLevel.bBusy	THEN
				IF fbSetPowerOnLevel.bError	THEN
					nStep	:= 900;
				ELSE	
					nStep	:= 50;
				END_IF
			END_IF
		
	50	:	fbSetSystemFailureLevel(bStart:=TRUE);
			IF NOT fbSetSystemFailureLevel.bBusy	THEN
				IF fbSetSystemFailureLevel.bError	THEN
					nStep	:= 900;
				ELSE	
					nStep	:= 60;
				END_IF
			END_IF
		
	60	:	fbSetFadeTime(bStart:=TRUE, );
			IF NOT fbSetFadeTime.bBusy	THEN
				IF fbSetFadeTime.bError	THEN
					nStep	:= 900;
				ELSE	
					nStep	:= 70;
				END_IF
			END_IF
		
	70	:	fbSetExtendedFadeTime(bStart:=TRUE);
			IF NOT fbSetExtendedFadeTime.bBusy	THEN
				IF fbSetExtendedFadeTime.bError	THEN
					nStep	:= 900;
				ELSE	
					nStep	:= 80;
				END_IF
			END_IF
		
	80	:	fbSetFadeRate(bStart:=TRUE);
			IF NOT fbSetFadeRate.bBusy	THEN
				IF fbSetFadeRate.bError	THEN
					nStep	:= 900;
				ELSE	
					nStep	:= 110;
				END_IF
			END_IF
		
	110	:	fbStopQuiescentMode(bStart:=TRUE);
			IF NOT fbStopQuiescentMode.bBusy	THEN
				IF fbStopQuiescentMode.bError	THEN
					nStep	:= 900;
				ELSE	
					nStep	:= 800;
				END_IF
			END_IF
			
	800	: 	// Completed
			bInitializationDone	:= TRUE;
			nStep	:= 0;
			
	900	: 	// Error
			bInitializationErr	:= TRUE;
			nStep	:= 0;
	
END_CASE

bInitializing	:= (nStep>0);
END_METHOD

{attribute 'hide'}
METHOD PROTECTED CheckGroupRefDev : BOOL	// Check if the reference device belongs to the addressed group
VAR_INPUT
	bEn				: BOOL;
END_VAR             
VAR_INST            
	nStep			: INT;
	fbQueryGroups	: FB_DALI102QueryGroups(0);
	_nAdr			: BYTE	:= 255;
	_nAdrRefDev		: BYTE	:= 255;
END_VAR             
VAR                 
	sErrorMessage	: T_MaxString ;
END_VAR
fbQueryGroups.ipDALICommunication	:= THIS^.ipDALICommunication;
fbQueryGroups.nAddress				:= THIS^.nAdrRefDev; 
fbQueryGroups.eAddressType			:= Tc3_DALI.E_DALIAddressType.Short; 
fbQueryGroups.eCommandPriority		:= Tc3_DALI.E_DALICommandPriority.Low;


IF NOT bEn	THEN
	RETURN;
END_IF

{region 'check membership of reference-device'}		
//+++++++++++ check membership of reference-device +++++++++++

 
IF 				(THIS^.eAdrType = Tc3_DALI.E_DALIAddressType.Group) 						// check group-membership of reference-device
	AND_THEN	((_nAdr <> THIS^.nAdr) OR_ELSE (_nAdrRefDev <> THIS^.nAdrRefDev))	THEN	// do it only if group-number has changed or reference-device has changed, which is definitely the case at PLC-start
	nStep		:= 10;
	_nAdr		:= THIS^.nAdr;
	_nAdrRefDev	:= THIS^.nAdrRefDev;
END_IF	

CASE nStep	OF
	
	0	: 	// Idle
			
	10	:	// Start	
			fbQueryGroups(bStart	:= TRUE);

			IF (NOT fbQueryGroups.bBusy)  THEN	
				IF 	fbQueryGroups.bError	THEN			// Query Groups Error is also an indicator of wrong reference-device
					sErrorMessage	:= CONCAT('Reference device #', TO_STRING(THIS^.nAdrRefDev)); 
					sErrorMessage	:= CONCAT(sErrorMessage, ' may not exist, group #'); 
					sErrorMessage	:= CONCAT(sErrorMessage, TO_STRING(THIS^.nAdr)); 
						 
					THIS^.fbLogMsgReferenceDevice.Show(ADSLOG_MSGTYPE_ERROR, 'DALI-error QueryGroups', sErrorMessage, FALSE); 	// assembled message
						 
				ELSIF ( TO_WORD((EXPT(2,(THIS^.nAdr)))) AND fbQueryGroups.nGroups) =	0	THEN	// Reference-device does not belong to the addressed group
					sErrorMessage	:= CONCAT('Reference device #', TO_STRING(THIS^.nAdrRefDev)); 
					sErrorMessage	:= CONCAT(sErrorMessage, ' does not belong to group #'); 
					sErrorMessage	:= CONCAT(sErrorMessage, TO_STRING(THIS^.nAdr)); 
					 
					THIS^.fbLogMsgReferenceDevice.Show(ADSLOG_MSGTYPE_ERROR, 'DALI-error reference-device of group ', sErrorMessage, FALSE); 	// assembled message
	 			END_IF	
					 
				THIS^.fbLogMsgReferenceDevice.Reset();
				fbQueryGroups(bStart:= FALSE);
				nStep	:= 0; 
			END_IF                     					
END_CASE
{endregion}
END_METHOD

{attribute 'hide'}
METHOD PROTECTED GetAdressInfo : T_MaxString
VAR
	sAdressInfo		: T_MaxString ;
END_VAR
CASE THIS^.eAdrType	OF
	Tc3_DALI.E_DALIAddressType.Short:
		sAdressInfo	:= CONCAT('#', TO_STRING(THIS^.nAdr)); 
		sAdressInfo	:= CONCAT(sAdressInfo, ', short-addressed'); 
	Tc3_DALI.E_DALIAddressType.Group:
		sAdressInfo	:= CONCAT('#', TO_STRING(THIS^.nAdrRefDev)); 
		sAdressInfo	:= CONCAT(sAdressInfo, ' of group #'); 
		sAdressInfo	:= CONCAT(sAdressInfo, TO_STRING(THIS^.nAdr)); 
	Tc3_DALI.E_DALIAddressType.Broadcast:
		sAdressInfo	:= CONCAT('#', TO_STRING(THIS^.nAdrRefDev)); 
		sAdressInfo	:= CONCAT(sAdressInfo, ', broadcast-call'); 			   
END_CASE

GetAdressInfo	:= sAdressInfo;
END_METHOD

{attribute 'hide'}
METHOD PROTECTED GetLightVal : BOOL
VAR_INPUT
	bEn				: BOOL;
END_VAR             
VAR_INST            
	ftEnable			: F_TRIG;
	nStep				: INT;
	fbQueryLgtVal		: FB_DALI102QueryActualLevel(0);
	tonQuery			: TON;
	tQuery				: TIME;
END_VAR
VAR
	sAdressInfo			: T_MaxString ;
	sLineInfo			: T_MaxString ;
	sErrorMessage		: T_MaxString ;
END_VAR
fbQueryLgtVal.ipDALICommunication	:= THIS^.ipDALICommunication;
fbQueryLgtVal.nAddress				:= THIS^.nAdrRefDev;
fbQueryLgtVal.eAddressType			:= Tc3_DALI.E_DALIAddressType.Short;
fbQueryLgtVal.eCommandPriority		:= Tc3_DALI.E_DALICommandPriority.Low;

ftEnable(CLK	:= bEn);

IF ftEnable.Q	THEN
	fbQueryLgtVal			(bStart := FALSE);
	nStep					:= 0;
	THIS^.bGetLightValBusy	:= FALSE;
	tonQuery				(IN:=FALSE);
	THIS^.fbLogMsgGetLightValCmdErr.Reset();	
END_IF

IF NOT bEn	THEN
	RETURN;
END_IF

{region 'query light level'}	 
//+++++++++++ query light level +++++++++++
IF NOT THIS^.bInhibit	THEN	 
	tQuery	:= F_BA_UdiToTiSec(THIS^.nPrdQueryLgtVal);
ELSE		 
	tQuery	:= F_BA_UdiToTiSec(THIS^.nPrdQueryLgtVal_Fast);
END_IF		 
	 
tonQuery(IN:= (NOT tonQuery.Q AND NOT THIS^.bGetLightValBusy), PT:= tQuery);
	 
IF NOT THIS^.bGetLightValBusy	THEN
	IF tonQuery.Q	THEN
		nStep	:= 10;
	END_IF
END_IF	

CASE nStep	OF
	
	0	: 	// Idle
			
	10	:	// Start	
			fbQueryLgtVal( bStart	:= TRUE);
								 
			IF (NOT fbQueryLgtVal.bBusy) THEN
				IF	fbQueryLgtVal.bError THEN 
						 
					sAdressInfo	:= 	 THIS^.GetAdressInfo();
					sLineInfo	:= 	 THIS^.GetLineInfo();
						 
					CASE THIS^.eAdrType	OF																								// address-specific part of message
						Tc3_DALI.E_DALIAddressType.Short:
							sErrorMessage	:= CONCAT('Addressed device: ', sAdressInfo);
						Tc3_DALI.E_DALIAddressType.Group, Tc3_DALI.E_DALIAddressType.Broadcast:
							sErrorMessage	:= CONCAT('Reference device: ', sAdressInfo); 
					END_CASE
						 
					sErrorMessage	:= CONCAT(sErrorMessage, ','); 
					sErrorMessage	:= CONCAT(sErrorMessage, sLineInfo); 																// DALI-line-specific part of message
						 
					sErrorMessage	:= CONCAT(sErrorMessage, ', MessageId: ');  														// Message Id as mentioned in the event-logger
					sErrorMessage	:= CONCAT(sErrorMessage, TO_STRING(fbQueryLgtVal.ipResultMessage.nEventId)); 
						 
					THIS^.fbLogMsgGetLightValCmdErr.Show(ADSLOG_MSGTYPE_ERROR, 'DALI-error: QueryLightLevel', sErrorMessage, FALSE); 	// assembled message
				ELSE
					THIS^.fbLogMsgGetLightValCmdErr.Reset();	
					THIS^.nActlLgtVal:= fbQueryLgtVal.nActualLevel;
					THIS^.fActlLgtVal	:= TO_REAL(Tc3_DALI.DALI_TO_PERCENT(THIS^.nActlLgtVal));
				END_IF
				fbQueryLgtVal(bStart := FALSE);   
				nStep		:= 0; 
			END_IF                     					
	
END_CASE
	 
THIS^.bGetLightValBusy		:= (nStep <> 0);
THIS^.bGetLightValErr		:= fbQueryLgtVal.bError;
{endregion}
END_METHOD

{attribute 'hide'}
METHOD PROTECTED GetLineInfo : STRING(255)
VAR
	sLineInfo		: T_MaxString ;
	sAdressInfo		: T_MaxString ;
END_VAR
sLineInfo	:= CONCAT((' DALI-line: '), (THIS^.ipDALICommunication.GetInstancePath()));

GetLineInfo	:= sLineInfo;
END_METHOD

{attribute 'hide'}
METHOD PROTECTED SetLightVal : BOOL
VAR_INPUT
	bEn					: BOOL;
	fLgtVal				: REAL;							// 1..100%
END_VAR
VAR_INST
	_fLgtVal			: REAL;							// 1..100%
	ftEnable			: F_TRIG;
	nStep				: INT;
	fbSetLgtVal			: FB_DALI102DirectArcPowerControl(0);
	nLgtVal				: BYTE;							// 0..254
	bInitLgtVal			: BOOL;
	rtZero				: R_TRIG;
	bSetZero			: BOOL;	
END_VAR
VAR
	sLineInfo			: T_MaxString ;
	sErrorMessage		: T_MaxString ;
END_VAR
fbSetLgtVal.ipDALICommunication	:= THIS^.ipDALICommunication;
fbSetLgtVal.nAddress			:= THIS^.nAdr;
fbSetLgtVal.eAddressType		:= THIS^.eAdrType;
fbSetLgtVal.eCommandPriority	:= Tc3_DALI.E_DALICommandPriority.MiddleHigh;

ftEnable(CLK	:= bEn);

IF ftEnable.Q	THEN
	fbSetLgtVal(bStart		:= FALSE);   
	nStep					:= 0;
	THIS^.bSetLightValBusy	:= FALSE;
	THIS^.nActlLgtVal		:= 0;
	rtZero	(CLK := bEn);
	THIS^.fbLogMsSetLightValCmdErr.Reset();	
END_IF

IF NOT bEn	THEN
	RETURN;
END_IF

fLgtVal				:= LIMIT(0, fLgtVal,100);
THIS^.nHysLgtVal 	:= LIMIT(2, THIS^.nHysLgtVal, 50);	
nLgtVal				:= Tc3_DALI.PERCENT_TO_DALI (fLgtVal);

IF	nLgtVal > 0	THEN
	nLgtVal	 	:= LIMIT(nMinLevel, nLgtVal, nMaxLevel);
END_IF

{region 'set light level'}
//+++++++++++ set light level +++++++++++

rtZero(CLK:= (nLgtVal=0));
IF rtZero.Q	THEN
	bSetZero	:= TRUE;
END_IF	

IF NOT THIS^.bSetLightValBusy	THEN
	IF NOT bInitLgtVal OR  (ABS(TO_REAL(THIS^.nActlLgtVal)-TO_REAL(nLgtVal))>= TO_REAL(THIS^.nHysLgtVal/2))	THEN
		bInitLgtVal	:= TRUE;
		nStep	:= 10;	
	ELSIF	bSetZero		THEN	// if the hysteresis does not let the light be set to 0, then it will be explicitely done here
		nStep	:= 15;
	END_IF
END_IF	

CASE nStep	OF
	
	0	: 	// Idle
			
	10	: 	// Start
			fbSetLgtVal(	bStart			:= TRUE,
							nArcPowerLevel	:= nLgtVal);  
			nStep		:= 20;

	15	: 	// Set explicitely to zero
			fbSetLgtVal(	bStart			:= TRUE,
							nArcPowerLevel	:= 0);
			nLgtVal		:= 0;
			bSetZero	:= FALSE;
			nStep		:= 20;
			
	20	:	// Wait  
			fbSetLgtVal();
				 
			IF (NOT fbSetLgtVal.bBusy) THEN	
				IF	fbSetLgtVal.bError 	THEN
						 
					sLineInfo	:= 	 THIS^.GetLineInfo();
						 
					CASE THIS^.eAdrType	OF																								// address-specific part of message
						Tc3_DALI.E_DALIAddressType.Short:
							sErrorMessage	:= CONCAT('Addressed single-device: #', TO_STRING(THIS^.nAdr));
						Tc3_DALI.E_DALIAddressType.Group:
							sErrorMessage	:= CONCAT('Addressed group: #', TO_STRING(THIS^.nAdr));
						Tc3_DALI.E_DALIAddressType.Broadcast:
							sErrorMessage	:= 'Broadcast'; 
					END_CASE
						 
					sErrorMessage	:= CONCAT(sErrorMessage, ','); 
					sErrorMessage	:= CONCAT(sErrorMessage, sLineInfo); 																// DALI-line-specific part of message
						 
					sErrorMessage	:= CONCAT(sErrorMessage, ', MessageId: ');   														// Message Id as mentioned in the event-logger
					sErrorMessage	:= CONCAT(sErrorMessage, TO_STRING(fbSetLgtVal.ipResultMessage.nEventId)); 
						 
					THIS^.fbLogMsgGetLightValCmdErr.Show(ADSLOG_MSGTYPE_ERROR, 'DALI-error: SetLightLevel', sErrorMessage, FALSE); 	// assembled message
						 
				ELSE
					THIS^.fbLogMsSetLightValCmdErr.Reset();	
					THIS^.nActlLgtVal := nLgtVal;						// predicted actual value by successful command 
					THIS^.fActlLgtVal := TO_REAL(Tc3_DALI.DALI_TO_PERCENT(THIS^.nActlLgtVal));
				END_IF
				fbSetLgtVal(bStart	:= FALSE);   
				nStep		:= 0; 
			END_IF                                                 
END_CASE
	 
THIS^.bSetLightValBusy		:= (nStep <> 0);
THIS^.bSetLightValErr		:= fbSetLgtVal.bError;
{endregion}
END_METHOD

END_FUNCTION_BLOCK

// ---- Templates/POUs/Trade/RoomAutomation/Common/Sensors/FB_BA_BrightnessPresenceDALI.TcPOU
{region '#Template'}
	{attribute 'Version' := '5.1.0.0'}
	{attribute 'Tags' := '"LCID": "1031", "Text": "RA, Sensoren, DALI, Präsenzmelder"'}
	{attribute 'Tags' := '"LCID": "1033", "Text": "RA, Sensors, DALI, presence-detection"'}
	{attribute 'Description' := '"LCID": "1031", "Text": "Template DALI Präsenzmelder"'}
	{attribute 'Description' := '"LCID": "1033", "Text": "Template DALI presence-detection"'}
{endregion}
FUNCTION_BLOCK FB_BA_BrightnessPresenceDALI EXTENDS FB_BA_Ext_BrightnessPresence_Base

VAR_INPUT
	bEn						: BOOL;			// FB-enable
	bInitialize				: BOOL;			// initialize with DALI-parameters
	bResetPresence			: BOOL;			// reset internal PLC-programmed delay-timer and trigger bRstSwi
	{attribute 'parameterUnit':= 's'}
	nPrdQueryBrtns			: UDINT	:= 1;	// [s] query interval of brightness
END_VAR
VAR_OUTPUT
	bPresence				: BOOL;			// presence detected
	bPresenceDelayActive	: BOOL;			// presence detection is FALSE, output bPresence is only set by delay-timer 
	bRstSwi					: BOOL;			// reset manual switch especially for sunblinds (presence for sunblinds differs between thermoautomatic and sunprotection)
	fBrightness				: REAL;			// brightness value
	bInitializing			: BOOL;			// device is being initialized
	bErr					: BOOL;			// error
END_VAR
VAR_INPUT CONSTANT PERSISTENT
	nAdr					: BYTE;	
	nInstancePresence		: BYTE;	
	nInstanceBrightness		: BYTE;	
	nResBrtns				: BYTE;			// manufacturers specific resolution	
	ipDALICommunication		: Tc3_DALI.I_DALICommunication;
END_VAR
VAR_INPUT CONSTANT
	BrightnessPresenceSns	: FB_BA_BrtnsPrcDALI;
	PresenceDelay			: FB_BA_PresenceMonitoring;		
	Brightness				: FB_BA_AI_Raw;
	Presence				: FB_BA_BI_Raw;		
END_VAR
VAR
END_VAR

SUPER^(); // FB_BA_Ext_BrightnessPresence_Base
BrightnessPresenceSns(
    bEn := bEn,
    bInitialize := bInitialize_In OR bInitialize,
    nPrdQueryBrtns := nPrdQueryBrtns,
    nAdr := nAdr,
    nInstPrc := nInstancePresence,
    nInstBrtns := nInstanceBrightness,
    nResBrtns := nResBrtns,
    ipDALICommunication := ipDALICommunication); // FB_BA_BrtnsPrcDALI
bInitializing := BrightnessPresenceSns.bInitializing;
bErr := BrightnessPresenceSns.bErr;
PresenceDelay(
    bPresence := BrightnessPresenceSns.bPrc,
    bRstDelayTimer := bResetPresence,
    bRstManMod := bResetPresence); // FB_BA_PresenceMonitoring
bRstSwi := PresenceDelay.bRstSwi;
bPresence := PresenceDelay.bPresenceState;
bPresenceDelayActive := PresenceDelay.bPresenceDelayActive;
Presence(bRawVal := PresenceDelay.bPresenceState); // FB_BA_BI_Raw
Brightness(nRawState := 0, nRawVal := TO_INT(BrightnessPresenceSns.nBrtns)); // FB_BA_AI_Raw
fBrightness := Brightness.fPresentValue;

METHOD FB_init : BOOL
VAR_INPUT
	bInitRetains : BOOL; // if TRUE; the retain variables are initialized (warm start / cold start)
	bInCopyCode : BOOL;  // if TRUE; the instance afterwards gets moved into the copy code (online change)
END_VAR
BrightnessPresenceSns.nDeadtime			:= 2;				// Dead-time-timer as multiple of 50ms
BrightnessPresenceSns.nHold				:= 5;				// Hold-timer as multiple of 10s, a "0" means 1s
BrightnessPresenceSns.nReport			:= 60;				// Report-timer in s BrightnesPresenceSns

PresenceDelay.nDlyPrc					:= 600;				// Presence delay [s] (in addition to the DALI-hold-timer!)			
	
// Presence-detection (delayed) // Präsenzmeldung ausschaltverzögert	
Presence.iParent						:= THIS^;								
Presence.iLabel							:= LblFun_Status;
Presence.ePolarity						:= E_BA_Polarity.eNormal;
Presence.sActiveText 					:= txtEvent_Occupied;
Presence.sInactiveText 					:= txtEvent_NotOccupied;
Presence.nEventClassID					:= EC_ID.NC80;
Presence.stTimeDelay.nToNormal			:= 0;
Presence.stTimeDelay.nToAbnormal		:= 0;
Presence.bAlarmValue					:= TRUE;
Presence.aEventTransitionText[1]		:= txtEvent_Triggered;
Presence.aEventTransitionText[2]		:= txtEvent_Error;
Presence.aEventTransitionText[3]		:= txtEvent_Normal;
Presence.bEventDetectionEnable			:= TRUE;
Presence.eEnPlantLock					:= E_BA_LockPriority.eNoLock;

// Brightness scaled // skalierte Helligkeit
Brightness.iParent						:= THIS^;		
Brightness.iLabel						:= LblFun_MeasuredValue;
Brightness.eUnit						:= E_BA_Unit.eLight_Luxes;
Brightness.fResolution 					:= 1; // in case, the manufacturer supplies a lux-value
Brightness.fScaleOffset 				:= 0; 	
Brightness.fCOVIncrement				:= BA2_Param.fDefCOVIncrement;
Brightness.nEventClassID				:= EC_ID.NC80;
Brightness.stTimeDelay.nToNormal		:= BA2_Param.nDefTimeDelay_ToNormal;
Brightness.stTimeDelay.nToAbnormal		:= BA2_Param.nDefTimeDelay_ToAbnormal;
Brightness.stHighLimit.bEnable			:= FALSE;
Brightness.stHighLimit.fValue			:= 0.0;		
Brightness.stLowLimit.bEnable			:= FALSE;
Brightness.stLowLimit.fValue			:= 0.0;
Brightness.fLimitDeadband 				:= BA2_Param.fDefLimitDeadband;
Brightness.aEventTransitionText[1]		:= txtEvent_Exceeded;
Brightness.aEventTransitionText[2]		:= txtEvent_Disturb;
Brightness.aEventTransitionText[3]		:= txtEvent_Normal;
Brightness.bEventDetectionEnable		:= TRUE;
Brightness.eEnPlantLock					:= E_BA_LockPriority.eNoLock;
END_METHOD

END_FUNCTION_BLOCK

// ---- Templates/POUs/Trade/RoomAutomation/Communication/FB_BA_AdsComServer_Room.TcPOU
{region '#Template'}
	{attribute 'Version' := '5.1.0.0'}
	{attribute 'Tags' := '"LCID": "1031", "Text": "Gebäudeautomation, Kommunikation, Server, Client, Publisher, Subscriber"'}
	{attribute 'Tags' := '"LCID": "1033", "Text": "Building automation, Communication, Server, Client, Publisher, Subscriber"'}
	{attribute 'Using' := '"Type": "Template", "URI": "Site"'}
	{attribute 'Description' := '"LCID": "1031", "Text": "Server Datenkommunikation"'}
	{attribute 'Description' := '"LCID": "1033", "Text": "Server data communication"'}
{endregion}

FUNCTION_BLOCK FB_BA_AdsComServer_Room
VAR_INPUT CONSTANT
  	BuildingEnergyLevel		: FB_BA_RawPublisher;
	BuildingSpRmT			: FB_BA_RawPublisher;
	BuildingLighting		: FB_BA_RawPublisher;
END_VAR

BuildingEnergyLevel(xData := Site.eBuildingEnergyLevel); // FB_BA_RawPublisher
BuildingSpRmT(xData := Site.stBuildingSpRmT); // FB_BA_RawPublisher
BuildingLighting(xData := Site.stBuildingLighting); // FB_BA_RawPublisher

END_FUNCTION_BLOCK

// ---- Templates/POUs/Trade/RoomAutomation/HeatingCooling/[Internal]/FB_BA_Ext_HeatCoolBase.TcPOU
{region '#Template'}
	{attribute 'Version' := '5.0.0.0'}
	{attribute 'Tags' := '"LCID": "1031", "Text": "RA, Sunprotection, Sunblind, Zone"'}
	{attribute 'Tags' := '"LCID": "1033", "Text": "RA, Sunprotection, Sunblind, Zone"'}
	{attribute 'Using' := '"Type": "Template", "URI": "ST_BA_Facade"'}
	{attribute 'Description' := '"LCID": "1031", "Text": "Sonnenschutzlogik interner Baustein"'}
	{attribute 'Description' := '"LCID": "1033", "Text": "Sunblind-logic inernal function)"'}
{endregion}
FUNCTION_BLOCK FB_BA_Ext_HeatCoolBase EXTENDS FB_BA_View
VAR		
	{attribute 'BaParam.Title.DE' := 'Raumtemperaturannpassung'}
	{attribute 'BaParam.Title.EN' := 'Room temperature adjustment'}
	{attribute 'BaParam.Access.Write' := 'Basic'}
	fRmTAdj_In				: REAL;
	{attribute 'BaParam.Title.DE' := 'Rückmeldung Raumtemperaturannpassung'}
	{attribute 'BaParam.Title.EN' := 'Feedback room temperature adjustment'}
	{attribute 'BaParam.Access.Write' := 'Locked'}
	{attribute 'BaParam.Access.Read' := 'Guest'}
	fRmTAdj_Out				: REAL;
	{attribute 'BaParam.Title.DE' := 'Raumtemperaturannpassung Bereich'}
	{attribute 'BaParam.Title.EN' := 'Temperature adjust range'}
	{attribute 'BaParam.Access.Write' := 'Locked'}
	{attribute 'BaParam.Access.Read' := 'Guest'}
	fRmTAdjLimit_Out		: REAL;
	{attribute 'BaParam.Title.DE' := 'Raumtemperatur'}
	{attribute 'BaParam.Title.EN' := 'Room temperature'}
	{attribute 'BaParam.Access.Write' := 'Locked'}
	{attribute 'BaParam.Access.Read' := 'Guest'}
	fRmT_Out				: REAL;
	{attribute 'BaParam.Title.DE' := 'Sollwert Heizen'}
	{attribute 'BaParam.Title.EN' := 'Setpoint heating'}
	{attribute 'BaParam.Access.Write' := 'Locked'}
	{attribute 'BaParam.Access.Read' := 'Guest'}
	fSPHtg_Out				: REAL;	
	{attribute 'BaParam.Title.DE' := 'Sollwert Kühlen'}
	{attribute 'BaParam.Title.EN' := 'Setpoint cooling'}
	{attribute 'BaParam.Access.Write' := 'Locked'}
	{attribute 'BaParam.Access.Read' := 'Guest'}
	fSPCol_Out				: REAL;		
	{attribute 'BaParam.Title.DE' := 'Reglerausgang Heizen'}
	{attribute 'BaParam.Title.EN' := 'Control value heating'}
	{attribute 'BaParam.Access.Write' := 'Locked'}
	{attribute 'BaParam.Access.Read' := 'Guest'}
	fCtrlValHtg_Out			: REAL;		
	{attribute 'BaParam.Title.DE' := 'Reglerausgang Kühlen'}
	{attribute 'BaParam.Title.EN' := 'Control value cooling'}
	{attribute 'BaParam.Access.Write' := 'Locked'}
	{attribute 'BaParam.Access.Read' := 'Guest'}
	fCtrlValCol_Out			: REAL;		
	{attribute 'BaParam.Title.DE' := 'Aktuelles Raumenergieniveau'}
	{attribute 'BaParam.Title.EN' := 'Actual room energy level'}
	{attribute 'BaParam.Access.Write' := 'Locked'}
	{attribute 'BaParam.Access.Read' := 'Guest'}
	eActualEnergyLevel_Out	: E_BA_EnergyLvlEx;
	{attribute 'BaParam.Title.DE' := 'Fehler'}
	{attribute 'BaParam.Title.EN' := 'Error'}
	{attribute 'BaParam.Access.Write' := 'Locked'}
	{attribute 'BaParam.Access.Read' := 'Guest'}
	bErr_Out				: BOOL;
END_VAR

VAR
	_fRmTAdj_Out			: REAL;
END_VAR

SUPER^();

IF (_fRmTAdj_Out<>fRmTAdj_Out)	THEN
	fRmTAdj_In	:= fRmTAdj_Out;		// set EXT-setpoint to actual resulting setpont in the template if this value has changed
END_IF

_fRmTAdj_Out:=fRmTAdj_Out;

END_FUNCTION_BLOCK

// ---- Templates/POUs/Trade/RoomAutomation/Lighting/Functions/Zone/FB_BA_LightGroupConstant.TcPOU
{region '#Template'}
	{attribute 'Version' := '5.0.0.0'}
	{attribute 'Tags' := '"LCID": "1031", "Text": "RA, Beleuchtung, Anwenderfunktionen, Konstantlicht"'}
	{attribute 'Tags' := '"LCID": "1033", "Text": "RA, Lighting, User-functions, constant light control"'}
	{attribute 'Using' := '"Type": "Template", "URI": "ST_BA_LightActuatorFeedback"'}
	{attribute 'Description' := '"LCID": "1031", "Text": "Beleuchtung Konstantlichtregelung"'}
	{attribute 'Description' := '"LCID": "1033", "Text": "Lighting constant light control"'}
{endregion}
FUNCTION_BLOCK FB_BA_LightGroupConstant EXTENDS FB_BA_Ext_LightConstCtrl
VAR_INPUT
	bManualSwitch			: BOOL;
	bOn						: BOOL;
	bOff					: BOOL;
	bResetRoomFunction		: BOOL;			// inactivates the whole function: control-mode AND manual-mode
	bPresence				: BOOL;
	fBrightness				: REAL;
	                        
	stAreaLighting			: ST_BA_Lighting;
	stScene					: ST_BA_Lighting;
	stReferenceFeedback		: ST_BA_LightActuatorFeedback;
	                        
END_VAR                     
                            
VAR_OUTPUT                  
	stLighting				: ST_BA_Lighting;
	bAdjusting				: BOOL;				// This signal is to be used to poll the brightness faster in case of a fieldbus-based brightness-sensor
END_VAR

		
